LIN {X 0,Y 516.984,Z 233.939,A -85,B 0,C 180,E1 -5032.678,E2 -5032.678} C_VEL
LIN {X 0,Y 516.803,Z 243.028,A -85,B 0,C 180,E1 -5033.356,E2 -5033.356} C_VEL
LIN {X 0,Y 516.628,Z 250.94,A -85,B 0,C 180,E1 -5034.144,E2 -5034.144} C_VEL
LIN {X 0,Y 516.608,Z 257.035,A -85,B 0,C 180,E1 -5034.927,E2 -5034.927} C_VEL
LIN {X 0,Y 516.481,Z 261.852,A -85,B 0,C 180,E1 -5035.708,E2 -5035.708} C_VEL
LIN {X 0,Y 516.468,Z 265.615,A -85,B 0,C 180,E1 -5036.489,E2 -5036.489} C_VEL
LIN {X 0,Y 516.284,Z 269.666,A -85,B 0,C 180,E1 -5037.66,E2 -5037.66} C_VEL
LIN {X 0,Y 516.212,Z 271.428,A -85,B 0,C 180,E1 -5038.44,E2 -5038.44} C_VEL
LIN {X 0,Y 516.197,Z 272.491,A -85,B 0,C 180,E1 -5039.22,E2 -5039.22} C_VEL
LIN {X 0,Y 516.195,Z 272.884,A -85,B 0,C 180,E1 -5040,E2 -5040} C_VEL
LIN {X 0,Y 516.199,Z 272.616,A -85,B 0,C 180,E1 -5040.78,E2 -5040.78} C_VEL
LIN {X 0,Y 516.215,Z 271.681,A -85,B 0,C 180,E1 -5041.56,E2 -5041.56} C_VEL
LIN {X 0,Y 516.332,Z 268.959,A -85,B 0,C 180,E1 -5042.731,E2 -5042.731} C_VEL
LIN {X 0,Y 516.467,Z 266.206,A -85,B 0,C 180,E1 -5043.511,E2 -5043.511} C_VEL
LIN {X 0,Y 516.515,Z 261.551,A -85,B 0,C 180,E1 -5044.487,E2 -5044.487} C_VEL
LIN {X 0,Y 516.586,Z 256.656,A -85,B 0,C 180,E1 -5045.269,E2 -5045.269} C_VEL
LIN {X 0,Y 516.619,Z 250.449,A -85,B 0,C 180,E1 -5046.052,E2 -5046.052} C_VEL
LIN {X 0,Y 516.845,Z 242.132,A -85,B 0,C 180,E1 -5046.858,E2 -5046.858} C_VEL
LIN {X 0,Y 517.047,Z 233.07,A -85,B 0,C 180,E1 -5047.518,E2 -5047.518} C_VEL
LIN {X 0,Y 517.237,Z 222.858,A -85,B 0,C 180,E1 -5048.055,E2 -5048.055} C_VEL
LIN {X 0,Y 516.418,Z 214.88,A -85,B 0,C 180,E1 -5048.388,E2 -5048.388} C_VEL
LIN {X 0,Y 516.468,Z 207.091,A -85,B 0,C 180,E1 -5050.983,E2 -5050.983} C_VEL
LIN {X 0,Y 516.61,Z 197.576,A -85,B 0,C 180,E1 -5054.174,E2 -5054.174} C_VEL
LIN {X 0,Y 516.772,Z 188.041,A -85,B 0,C 180,E1 -5057.409,E2 -5057.409} C_VEL
LIN {X 0,Y 516.892,Z 179.78,A -85,B 0,C 180,E1 -5060.252,E2 -5060.252} C_VEL
LIN {X 0,Y 517.052,Z 171.31,A -85,B 0,C 180,E1 -5063.215,E2 -5063.215} C_VEL
LIN {X 0,Y 517.347,Z 161.729,A -85,B 0,C 180,E1 -5066.635,E2 -5066.635} C_VEL
LIN {X 0,Y 517.599,Z 153.467,A -85,B 0,C 180,E1 -5069.657,E2 -5069.657} C_VEL
LIN {X 0,Y 517.235,Z 149.681,A -85,B 0,C 180,E1 -5071.126,E2 -5071.126} C_VEL
LIN {X 0,Y 516.93,Z 148.099,A -85,B 0,C 180,E1 -5071.792,E2 -5071.792} C_VEL
LIN {X 0,Y 516.885,Z 148.104,A -85,B 0,C 180,E1 -5074.825,E2 -5074.825} C_VEL
LIN {X 0,Y 516.886,Z 148.103,A -85,B 0,C 180,E1 -5077.943,E2 -5077.943} C_VEL
LIN {X 0,Y 516.889,Z 148.101,A -85,B 0,C 180,E1 -5080.741,E2 -5080.741} C_VEL
LIN {X 0,Y 516.888,Z 148.102,A -85,B 0,C 180,E1 -5082.831,E2 -5082.831} C_VEL
LIN {X 0,Y 516.901,Z 148.1,A -85,B 0,C 180,E1 -5085.007,E2 -5085.007} C_VEL
LIN {X 0,Y 516.92,Z 148.097,A -85,B 0,C 180,E1 -5088.398,E2 -5088.398} C_VEL
LIN {X 0,Y 516.885,Z 148.103,A -85,B 0,C 180,E1 -5091.284,E2 -5091.284} C_VEL
LIN {X 0,Y 516.877,Z 148.104,A -85,B 0,C 180,E1 -5094.219,E2 -5094.219} C_VEL
LIN {X 0,Y 516.887,Z 148.104,A -85,B 0,C 180,E1 -5097.051,E2 -5097.051} C_VEL
LIN {X 0,Y 516.924,Z 148.188,A -85,B 0,C 180,E1 -5099.982,E2 -5099.982} C_VEL
LIN {X 0,Y 518.784,Z 157.254,A -85,B 0,C 180,E1 -5102.573,E2 -5102.573} C_VEL
LIN {X 0,Y 518.974,Z 160.749,A -85,B 0,C 180,E1 -5103.455,E2 -5103.455} C_VEL
LIN {X 0,Y 518.28,Z 171.627,A -85,B 0,C 180,E1 -5105.995,E2 -5105.995} C_VEL
LIN {X 0,Y 517.784,Z 182.925,A -85,B 0,C 180,E1 -5108.5,E2 -5108.5} C_VEL
LIN {X 0,Y 517.391,Z 194.575,A -85,B 0,C 180,E1 -5110.973,E2 -5110.973} C_VEL
LIN {X 0,Y 517.079,Z 207.5,A -85,B 0,C 180,E1 -5113.618,E2 -5113.618} C_VEL
LIN {X 0,Y 516.843,Z 220.945,A -85,B 0,C 180,E1 -5116.27,E2 -5116.27} C_VEL
LIN {X 0,Y 518.188,Z 232.011,A -85,B 0,C 180,E1 -5116.519,E2 -5116.519} C_VEL
LIN {X 0,Y 518.022,Z 244.633,A -85,B 0,C 180,E1 -5116.914,E2 -5116.914} C_VEL
LIN {X 0,Y 517.734,Z 256.944,A -85,B 0,C 180,E1 -5117.455,E2 -5117.455} C_VEL
LIN {X 0,Y 517.492,Z 268.95,A -85,B 0,C 180,E1 -5118.159,E2 -5118.159} C_VEL
LIN {X 0,Y 517.222,Z 280.568,A -85,B 0,C 180,E1 -5119.033,E2 -5119.033} C_VEL
LIN {X 0,Y 516.967,Z 289.07,A -85,B 0,C 180,E1 -5119.819,E2 -5119.819} C_VEL
LIN {X 0,Y 516.761,Z 297.894,A -85,B 0,C 180,E1 -5120.804,E2 -5120.804} C_VEL
LIN {X 0,Y 516.582,Z 306.427,A -85,B 0,C 180,E1 -5121.983,E2 -5121.983} C_VEL
LIN {X 0,Y 516.443,Z 312.245,A -85,B 0,C 180,E1 -5122.964,E2 -5122.964} C_VEL
LIN {X 0,Y 516.417,Z 317.908,A -85,B 0,C 180,E1 -5124.141,E2 -5124.141} C_VEL
LIN {X 0,Y 516.27,Z 322.337,A -85,B 0,C 180,E1 -5125.314,E2 -5125.314} C_VEL
LIN {X 0,Y 516.37,Z 324.685,A -85,B 0,C 180,E1 -5126.097,E2 -5126.097} C_VEL
LIN {X 0,Y 516.283,Z 326.587,A -85,B 0,C 180,E1 -5126.877,E2 -5126.877} C_VEL
LIN {X 0,Y 516.261,Z 328.016,A -85,B 0,C 180,E1 -5127.658,E2 -5127.658} C_VEL
LIN {X 0,Y 516.171,Z 329.652,A -85,B 0,C 180,E1 -5129.219,E2 -5129.219} C_VEL
LIN {X 0,Y 516.173,Z 329.879,A -85,B 0,C 180,E1 -5129.999,E2 -5129.999} C_VEL
LIN {X 0,Y 516.17,Z 329.664,A -85,B 0,C 180,E1 -5130.779,E2 -5130.779} C_VEL
LIN {X 0,Y 516.261,Z 328.056,A -85,B 0,C 180,E1 -5132.339,E2 -5132.339} C_VEL
LIN {X 0,Y 516.282,Z 326.64,A -85,B 0,C 180,E1 -5133.12,E2 -5133.12} C_VEL
LIN {X 0,Y 516.313,Z 323.669,A -85,B 0,C 180,E1 -5134.292,E2 -5134.292} C_VEL
LIN {X 0,Y 516.397,Z 319.639,A -85,B 0,C 180,E1 -5135.465,E2 -5135.465} C_VEL
LIN {X 0,Y 516.469,Z 313.671,A -85,B 0,C 180,E1 -5136.787,E2 -5136.787} C_VEL
LIN {X 0,Y 516.58,Z 306.611,A -85,B 0,C 180,E1 -5138.015,E2 -5138.015} C_VEL
LIN {X 0,Y 516.769,Z 298.141,A -85,B 0,C 180,E1 -5139.194,E2 -5139.194} C_VEL
LIN {X 0,Y 516.972,Z 289.385,A -85,B 0,C 180,E1 -5140.178,E2 -5140.178} C_VEL
LIN {X 0,Y 517.329,Z 278.602,A -85,B 0,C 180,E1 -5141.161,E2 -5141.161} C_VEL
LIN {X 0,Y 517.554,Z 267.789,A -85,B 0,C 180,E1 -5141.952,E2 -5141.952} C_VEL
LIN {X 0,Y 517.797,Z 256.672,A -85,B 0,C 180,E1 -5142.591,E2 -5142.591} C_VEL
LIN {X 0,Y 518.061,Z 244.294,A -85,B 0,C 180,E1 -5143.133,E2 -5143.133} C_VEL
LIN {X 0,Y 518.244,Z 232.51,A -85,B 0,C 180,E1 -5143.502,E2 -5143.502} C_VEL
LIN {X 0,Y 516.877,Z 220.782,A -85,B 0,C 180,E1 -5143.789,E2 -5143.789} C_VEL
LIN {X 0,Y 517.168,Z 205.909,A -85,B 0,C 180,E1 -5146.783,E2 -5146.783} C_VEL
LIN {X 0,Y 517.391,Z 194.717,A -85,B 0,C 180,E1 -5149.025,E2 -5149.025} C_VEL
LIN {X 0,Y 517.866,Z 180.952,A -85,B 0,C 180,E1 -5151.912,E2 -5151.912} C_VEL
LIN {X 0,Y 518.373,Z 167.18,A -85,B 0,C 180,E1 -5154.851,E2 -5154.851} C_VEL
LIN {X 0,Y 518.661,Z 157.378,A -85,B 0,C 180,E1 -5156.994,E2 -5156.994} C_VEL
LIN {X 0,Y 516.909,Z 148.101,A -85,B 0,C 180,E1 -5159.248,E2 -5159.248} C_VEL
LIN {X 0,Y 516.892,Z 148.102,A -85,B 0,C 180,E1 -5162.542,E2 -5162.542} C_VEL
LIN {X 0,Y 516.878,Z 148.101,A -85,B 0,C 180,E1 -5165.331,E2 -5165.331} C_VEL
LIN {X 0,Y 516.874,Z 148.101,A -85,B 0,C 180,E1 -5167.942,E2 -5167.942} C_VEL
LIN {X 0,Y 516.862,Z 148.106,A -85,B 0,C 180,E1 -5170.741,E2 -5170.741} C_VEL
LIN {X 0,Y 516.872,Z 148.102,A -85,B 0,C 180,E1 -5173.892,E2 -5173.892} C_VEL
LIN {X 0,Y 516.873,Z 148.103,A -85,B 0,C 180,E1 -5176.106,E2 -5176.106} C_VEL
LIN {X 0,Y 516.894,Z 148.101,A -85,B 0,C 180,E1 -5179.259,E2 -5179.259} C_VEL
LIN {X 0,Y 516.869,Z 148.101,A -85,B 0,C 180,E1 -5182.056,E2 -5182.056} C_VEL
LIN {X 0,Y 516.868,Z 148.099,A -85,B 0,C 180,E1 -5185.174,E2 -5185.174} C_VEL
LIN {X 0,Y 516.871,Z 148.102,A -85,B 0,C 180,E1 -5187.975,E2 -5187.975} C_VEL
LIN {X 0,Y 516.924,Z 148.097,A -85,B 0,C 180,E1 -5190.695,E2 -5190.695} C_VEL
LIN {X 0,Y 516.932,Z 148.093,A -85,B 0,C 180,E1 -5193.802,E2 -5193.802} C_VEL
LIN {X 0,Y 516.845,Z 148.102,A -85,B 0,C 180,E1 -5196.775,E2 -5196.775} C_VEL
LIN {X 0,Y 516.925,Z 148.095,A -85,B 0,C 180,E1 -5199.731,E2 -5199.731} C_VEL
LIN {X 0,Y 516.918,Z 148.098,A -85,B 0,C 180,E1 -5202.596,E2 -5202.596} C_VEL
LIN {X 0,Y 516.927,Z 148.093,A -85,B 0,C 180,E1 -5205.03,E2 -5205.03} C_VEL
LIN {X 0,Y 516.989,Z 148.085,A -85,B 0,C 180,E1 -5208.234,E2 -5208.234} C_VEL
LIN {X 0,Y 516.948,Z 148.092,A -85,B 0,C 180,E1 -5211.399,E2 -5211.399} C_VEL
LIN {X 0,Y 516.996,Z 148.084,A -85,B 0,C 180,E1 -5213.757,E2 -5213.757} C_VEL
LIN {X 0,Y 517.004,Z 148.083,A -85,B 0,C 180,E1 -5216.883,E2 -5216.883} C_VEL
LIN {X 0,Y 517.065,Z 148.076,A -85,B 0,C 180,E1 -5220,E2 -5220} C_VEL
LIN {X 0,Y 516.992,Z 148.087,A -85,B 0,C 180,E1 -5223.117,E2 -5223.117} C_VEL
LIN {X 0,Y 516.994,Z 148.089,A -85,B 0,C 180,E1 -5226.243,E2 -5226.243} C_VEL
LIN {X 0,Y 516.946,Z 148.095,A -85,B 0,C 180,E1 -5229.389,E2 -5229.389} C_VEL
LIN {X 0,Y 516.968,Z 148.088,A -85,B 0,C 180,E1 -5231.824,E2 -5231.824} C_VEL
LIN {X 0,Y 516.931,Z 148.092,A -85,B 0,C 180,E1 -5235.148,E2 -5235.148} C_VEL
LIN {X 0,Y 516.911,Z 148.098,A -85,B 0,C 180,E1 -5238.223,E2 -5238.223} C_VEL
LIN {X 0,Y 516.901,Z 148.097,A -85,B 0,C 180,E1 -5240.702,E2 -5240.702} C_VEL
LIN {X 0,Y 516.878,Z 148.102,A -85,B 0,C 180,E1 -5243.223,E2 -5243.223} C_VEL
LIN {X 0,Y 516.888,Z 148.102,A -85,B 0,C 180,E1 -5246.188,E2 -5246.188} C_VEL
LIN {X 0,Y 516.903,Z 148.099,A -85,B 0,C 180,E1 -5249.526,E2 -5249.526} C_VEL
LIN {X 0,Y 516.889,Z 148.099,A -85,B 0,C 180,E1 -5252.545,E2 -5252.545} C_VEL
LIN {X 0,Y 516.872,Z 148.1,A -85,B 0,C 180,E1 -5255.334,E2 -5255.334} C_VEL
LIN {X 0,Y 516.868,Z 148.105,A -85,B 0,C 180,E1 -5257.944,E2 -5257.944} C_VEL
LIN {X 0,Y 516.871,Z 148.098,A -85,B 0,C 180,E1 -5260.743,E2 -5260.743} C_VEL
LIN {X 0,Y 516.874,Z 148.102,A -85,B 0,C 180,E1 -5262.832,E2 -5262.832} C_VEL
LIN {X 0,Y 516.913,Z 148.099,A -85,B 0,C 180,E1 -5265.011,E2 -5265.011} C_VEL
LIN {X 0,Y 516.909,Z 148.099,A -85,B 0,C 180,E1 -5268.4,E2 -5268.4} C_VEL
LIN {X 0,Y 516.872,Z 148.1,A -85,B 0,C 180,E1 -5270.322,E2 -5270.322} C_VEL
LIN {X 0,Y 516.198,Z 148.185,A -85,B 0,C 180,E1 -5270.972,E2 -5270.972} C_VEL
LIN {X 0,Y 513.338,Z 148.54,A -85,B 0,C 180,E1 -5272.027,E2 -5272.027} C_VEL
LIN {X 0,Y 510.923,Z 148.842,A -85,B 0,C 180,E1 -5272.878,E2 -5272.878} C_VEL
LIN {X 0,Y 509.883,Z 148.972,A -85,B 0,C 180,E1 -5273.534,E2 -5273.534} C_VEL
LIN {X 0,Y 509.797,Z 148.981,A -85,B 0,C 180,E1 -5273.757,E2 -5273.757} C_VEL
LIN {X 0,Y 509.853,Z 148.978,A -85,B 0,C 180,E1 -5276.541,E2 -5276.541} C_VEL
LIN {X 0,Y 509.845,Z 148.976,A -85,B 0,C 180,E1 -5279.336,E2 -5279.336} C_VEL
LIN {X 0,Y 509.89,Z 148.971,A -85,B 0,C 180,E1 -5282.056,E2 -5282.056} C_VEL
LIN {X 0,Y 509.806,Z 148.983,A -85,B 0,C 180,E1 -5284.702,E2 -5284.702} C_VEL
LIN {X 0,Y 509.82,Z 148.977,A -85,B 0,C 180,E1 -5287.46,E2 -5287.46} C_VEL
LIN {X 0,Y 509.914,Z 148.97,A -85,B 0,C 180,E1 -5289.846,E2 -5289.846} C_VEL
LIN {X 0,Y 509.883,Z 148.975,A -85,B 0,C 180,E1 -5293.176,E2 -5293.176} C_VEL
LIN {X 0,Y 509.852,Z 148.974,A -85,B 0,C 180,E1 -5295.635,E2 -5295.635} C_VEL
LIN {X 0,Y 509.911,Z 148.967,A -85,B 0,C 180,E1 -5298.876,E2 -5298.876} C_VEL
LIN {X 0,Y 509.951,Z 148.964,A -85,B 0,C 180,E1 -5302.08,E2 -5302.08} C_VEL
LIN {X 0,Y 509.983,Z 148.959,A -85,B 0,C 180,E1 -5304.466,E2 -5304.466} C_VEL
LIN {X 0,Y 510.056,Z 148.949,A -85,B 0,C 180,E1 -5307.632,E2 -5307.632} C_VEL
LIN {X 0,Y 510.036,Z 148.956,A -85,B 0,C 180,E1 -5310.001,E2 -5310.001} C_VEL
LIN {X 0,Y 510.051,Z 148.949,A -85,B 0,C 180,E1 -5312.37,E2 -5312.37} C_VEL
LIN {X 0,Y 509.982,Z 148.959,A -85,B 0,C 180,E1 -5316.331,E2 -5316.331} C_VEL
LIN {X 0,Y 509.914,Z 148.97,A -85,B 0,C 180,E1 -5318.721,E2 -5318.721} C_VEL
LIN {X 0,Y 509.908,Z 148.971,A -85,B 0,C 180,E1 -5321.933,E2 -5321.933} C_VEL
LIN {X 0,Y 509.899,Z 148.973,A -85,B 0,C 180,E1 -5325.243,E2 -5325.243} C_VEL
LIN {X 0,Y 509.866,Z 148.976,A -85,B 0,C 180,E1 -5328.485,E2 -5328.485} C_VEL
LIN {X 0,Y 509.855,Z 148.974,A -85,B 0,C 180,E1 -5331.003,E2 -5331.003} C_VEL
LIN {X 0,Y 509.822,Z 148.983,A -85,B 0,C 180,E1 -5333.565,E2 -5333.565} C_VEL
LIN {X 0,Y 509.819,Z 148.977,A -85,B 0,C 180,E1 -5336.357,E2 -5336.357} C_VEL
LIN {X 0,Y 509.842,Z 148.979,A -85,B 0,C 180,E1 -5338.847,E2 -5338.847} C_VEL
LIN {X 0,Y 509.823,Z 148.98,A -85,B 0,C 180,E1 -5341.591,E2 -5341.591} C_VEL
LIN {X 0,Y 509.843,Z 148.976,A -85,B 0,C 180,E1 -5344.415,E2 -5344.415} C_VEL
LIN {X 0,Y 509.793,Z 148.983,A -85,B 0,C 180,E1 -5347.344,E2 -5347.344} C_VEL
LIN {X 0,Y 509.818,Z 148.983,A -85,B 0,C 180,E1 -5350.385,E2 -5350.385} C_VEL
LIN {X 0,Y 509.808,Z 148.98,A -85,B 0,C 180,E1 -5353.06,E2 -5353.06} C_VEL
LIN {X 0,Y 509.828,Z 148.98,A -85,B 0,C 180,E1 -5355.794,E2 -5355.794} C_VEL
LIN {X 0,Y 509.86,Z 148.977,A -85,B 0,C 180,E1 -5358.575,E2 -5358.575} C_VEL
LIN {X 0,Y 509.819,Z 148.979,A -85,B 0,C 180,E1 -5361.792,E2 -5361.792} C_VEL
LIN {X 0,Y 509.83,Z 148.977,A -85,B 0,C 180,E1 -5364.622,E2 -5364.622} C_VEL
LIN {X 0,Y 509.865,Z 148.977,A -85,B 0,C 180,E1 -5367.481,E2 -5367.481} C_VEL
LIN {X 0,Y 509.905,Z 149.045,A -85,B 0,C 180,E1 -5368.71,E2 -5368.71} C_VEL
LIN {X 0,Y 510.39,Z 153.219,A -85,B 0,C 180,E1 -5370.283,E2 -5370.283} C_VEL
LIN {X 0,Y 510.177,Z 162.264,A -85,B 0,C 180,E1 -5373.563,E2 -5373.563} C_VEL
LIN {X 0,Y 509.935,Z 170.358,A -85,B 0,C 180,E1 -5376.442,E2 -5376.442} C_VEL
LIN {X 0,Y 509.805,Z 179.405,A -85,B 0,C 180,E1 -5379.625,E2 -5379.625} C_VEL
LIN {X 0,Y 509.665,Z 188.47,A -85,B 0,C 180,E1 -5382.754,E2 -5382.754} C_VEL
LIN {X 0,Y 509.53,Z 196.847,A -85,B 0,C 180,E1 -5385.625,E2 -5385.625} C_VEL
LIN {X 0,Y 509.379,Z 206.394,A -85,B 0,C 180,E1 -5388.863,E2 -5388.863} C_VEL
LIN {X 0,Y 509.323,Z 214.658,A -85,B 0,C 180,E1 -5391.619,E2 -5391.619} C_VEL
LIN {X 0,Y 510.161,Z 224.625,A -85,B 0,C 180,E1 -5392.032,E2 -5392.032} C_VEL
LIN {X 0,Y 509.982,Z 234.394,A -85,B 0,C 180,E1 -5392.577,E2 -5392.577} C_VEL
LIN {X 0,Y 509.761,Z 243.417,A -85,B 0,C 180,E1 -5393.264,E2 -5393.264} C_VEL
LIN {X 0,Y 509.571,Z 251.31,A -85,B 0,C 180,E1 -5394.063,E2 -5394.063} C_VEL
LIN {X 0,Y 509.555,Z 257.394,A -85,B 0,C 180,E1 -5394.857,E2 -5394.857} C_VEL
LIN {X 0,Y 509.423,Z 262.208,A -85,B 0,C 180,E1 -5395.648,E2 -5395.648} C_VEL
LIN {X 0,Y 509.41,Z 265.977,A -85,B 0,C 180,E1 -5396.441,E2 -5396.441} C_VEL
LIN {X 0,Y 509.215,Z 270.043,A -85,B 0,C 180,E1 -5397.627,E2 -5397.627} C_VEL
LIN {X 0,Y 509.132,Z 271.812,A -85,B 0,C 180,E1 -5398.418,E2 -5398.418} C_VEL
LIN {X 0,Y 509.109,Z 272.882,A -85,B 0,C 180,E1 -5399.209,E2 -5399.209} C_VEL
LIN {X 0,Y 509.107,Z 273.28,A -85,B 0,C 180,E1 -5400,E2 -5400} C_VEL
LIN {X 0,Y 509.111,Z 273.015,A -85,B 0,C 180,E1 -5400.791,E2 -5400.791} C_VEL
LIN {X 0,Y 509.135,Z 272.081,A -85,B 0,C 180,E1 -5401.582,E2 -5401.582} C_VEL
LIN {X 0,Y 509.265,Z 269.368,A -85,B 0,C 180,E1 -5402.769,E2 -5402.769} C_VEL
LIN {X 0,Y 509.433,Z 264.916,A -85,B 0,C 180,E1 -5403.955,E2 -5403.955} C_VEL
LIN {X 0,Y 509.539,Z 259.653,A -85,B 0,C 180,E1 -5404.945,E2 -5404.945} C_VEL
LIN {X 0,Y 509.612,Z 254.178,A -85,B 0,C 180,E1 -5405.738,E2 -5405.738} C_VEL
LIN {X 0,Y 509.717,Z 247.409,A -85,B 0,C 180,E1 -5406.508,E2 -5406.508} C_VEL
LIN {X 0,Y 509.902,Z 239.278,A -85,B 0,C 180,E1 -5407.225,E2 -5407.225} C_VEL
LIN {X 0,Y 510.131,Z 230.408,A -85,B 0,C 180,E1 -5407.819,E2 -5407.819} C_VEL
LIN {X 0,Y 510.108,Z 221.392,A -85,B 0,C 180,E1 -5408.268,E2 -5408.268} C_VEL
LIN {X 0,Y 509.353,Z 215.03,A -85,B 0,C 180,E1 -5408.53,E2 -5408.53} C_VEL
LIN {X 0,Y 509.411,Z 207.298,A -85,B 0,C 180,E1 -5411.137,E2 -5411.137} C_VEL
LIN {X 0,Y 509.55,Z 198.944,A -85,B 0,C 180,E1 -5413.968,E2 -5413.968} C_VEL
LIN {X 0,Y 509.684,Z 190.62,A -85,B 0,C 180,E1 -5416.832,E2 -5416.832} C_VEL
LIN {X 0,Y 509.854,Z 182.264,A -85,B 0,C 180,E1 -5419.738,E2 -5419.738} C_VEL
LIN {X 0,Y 510.02,Z 173.92,A -85,B 0,C 180,E1 -5422.696,E2 -5422.696} C_VEL
LIN {X 0,Y 510.222,Z 165.574,A -85,B 0,C 180,E1 -5425.715,E2 -5425.715} C_VEL
LIN {X 0,Y 510.576,Z 157.23,A -85,B 0,C 180,E1 -5428.801,E2 -5428.801} C_VEL
LIN {X 0,Y 510.506,Z 152.507,A -85,B 0,C 180,E1 -5430.622,E2 -5430.622} C_VEL
LIN {X 0,Y 509.857,Z 148.98,A -85,B 0,C 180,E1 -5432.169,E2 -5432.169} C_VEL
LIN {X 0,Y 509.835,Z 148.981,A -85,B 0,C 180,E1 -5435.378,E2 -5435.378} C_VEL
LIN {X 0,Y 509.855,Z 148.978,A -85,B 0,C 180,E1 -5438.338,E2 -5438.338} C_VEL
LIN {X 0,Y 509.861,Z 148.978,A -85,B 0,C 180,E1 -5441.425,E2 -5441.425} C_VEL
LIN {X 0,Y 509.845,Z 148.98,A -85,B 0,C 180,E1 -5444.67,E2 -5444.67} C_VEL
LIN {X 0,Y 509.839,Z 148.979,A -85,B 0,C 180,E1 -5447.51,E2 -5447.51} C_VEL
LIN {X 0,Y 509.851,Z 148.978,A -85,B 0,C 180,E1 -5450.647,E2 -5450.647} C_VEL
LIN {X 0,Y 509.831,Z 148.982,A -85,B 0,C 180,E1 -5453.646,E2 -5453.646} C_VEL
LIN {X 0,Y 509.848,Z 148.98,A -85,B 0,C 180,E1 -5456.537,E2 -5456.537} C_VEL
LIN {X 0,Y 509.873,Z 149.1,A -85,B 0,C 180,E1 -5459.565,E2 -5459.565} C_VEL
LIN {X 0,Y 511.72,Z 157.754,A -85,B 0,C 180,E1 -5462.162,E2 -5462.162} C_VEL
LIN {X 0,Y 512.12,Z 161.356,A -85,B 0,C 180,E1 -5463.128,E2 -5463.128} C_VEL
LIN {X 0,Y 511.433,Z 171.788,A -85,B 0,C 180,E1 -5465.653,E2 -5465.653} C_VEL
LIN {X 0,Y 510.78,Z 184.859,A -85,B 0,C 180,E1 -5468.615,E2 -5468.615} C_VEL
LIN {X 0,Y 510.299,Z 199.961,A -85,B 0,C 180,E1 -5471.859,E2 -5471.859} C_VEL
LIN {X 0,Y 509.878,Z 215.321,A -85,B 0,C 180,E1 -5475.021,E2 -5475.021} C_VEL
LIN {X 0,Y 509.822,Z 220.716,A -85,B 0,C 180,E1 -5476.115,E2 -5476.115} C_VEL
LIN {X 0,Y 511.155,Z 233.061,A -85,B 0,C 180,E1 -5476.406,E2 -5476.406} C_VEL
LIN {X 0,Y 510.997,Z 245.969,A -85,B 0,C 180,E1 -5476.832,E2 -5476.832} C_VEL
LIN {X 0,Y 510.713,Z 257.682,A -85,B 0,C 180,E1 -5477.369,E2 -5477.369} C_VEL
LIN {X 0,Y 510.441,Z 269.393,A -85,B 0,C 180,E1 -5478.08,E2 -5478.08} C_VEL
LIN {X 0,Y 510.161,Z 279.855,A -85,B 0,C 180,E1 -5478.879,E2 -5478.879} C_VEL
LIN {X 0,Y 509.864,Z 290.385,A -85,B 0,C 180,E1 -5479.877,E2 -5479.877} C_VEL
LIN {X 0,Y 509.652,Z 298.879,A -85,B 0,C 180,E1 -5480.874,E2 -5480.874} C_VEL
LIN {X 0,Y 509.49,Z 307.166,A -85,B 0,C 180,E1 -5482.07,E2 -5482.07} C_VEL
LIN {X 0,Y 509.308,Z 314.019,A -85,B 0,C 180,E1 -5483.303,E2 -5483.303} C_VEL
LIN {X 0,Y 509.309,Z 319.096,A -85,B 0,C 180,E1 -5484.456,E2 -5484.456} C_VEL
LIN {X 0,Y 509.221,Z 323.171,A -85,B 0,C 180,E1 -5485.645,E2 -5485.645} C_VEL
LIN {X 0,Y 509.202,Z 326.178,A -85,B 0,C 180,E1 -5486.834,E2 -5486.834} C_VEL
LIN {X 0,Y 509.19,Z 327.617,A -85,B 0,C 180,E1 -5487.626,E2 -5487.626} C_VEL
LIN {X 0,Y 509.084,Z 329.262,A -85,B 0,C 180,E1 -5489.208,E2 -5489.208} C_VEL
LIN {X 0,Y 509.084,Z 329.492,A -85,B 0,C 180,E1 -5489.999,E2 -5489.999} C_VEL
LIN {X 0,Y 509.112,Z 328.668,A -85,B 0,C 180,E1 -5491.581,E2 -5491.581} C_VEL
LIN {X 0,Y 509.19,Z 327.67,A -85,B 0,C 180,E1 -5492.372,E2 -5492.372} C_VEL
LIN {X 0,Y 509.201,Z 326.247,A -85,B 0,C 180,E1 -5493.164,E2 -5493.164} C_VEL
LIN {X 0,Y 509.206,Z 323.267,A -85,B 0,C 180,E1 -5494.352,E2 -5494.352} C_VEL
LIN {X 0,Y 509.309,Z 319.223,A -85,B 0,C 180,E1 -5495.542,E2 -5495.542} C_VEL
LIN {X 0,Y 509.399,Z 313.075,A -85,B 0,C 180,E1 -5496.912,E2 -5496.912} C_VEL
LIN {X 0,Y 509.496,Z 306.149,A -85,B 0,C 180,E1 -5498.127,E2 -5498.127} C_VEL
LIN {X 0,Y 509.717,Z 297.628,A -85,B 0,C 180,E1 -5499.322,E2 -5499.322} C_VEL
LIN {X 0,Y 509.945,Z 288.829,A -85,B 0,C 180,E1 -5500.32,E2 -5500.32} C_VEL
LIN {X 0,Y 510.317,Z 277.992,A -85,B 0,C 180,E1 -5501.316,E2 -5501.316} C_VEL
LIN {X 0,Y 510.505,Z 267.095,A -85,B 0,C 180,E1 -5502.116,E2 -5502.116} C_VEL
LIN {X 0,Y 510.817,Z 254.81,A -85,B 0,C 180,E1 -5502.816,E2 -5502.816} C_VEL
LIN {X 0,Y 511.111,Z 241.903,A -85,B 0,C 180,E1 -5503.365,E2 -5503.365} C_VEL
LIN {X 0,Y 511.158,Z 231.034,A -85,B 0,C 180,E1 -5503.693,E2 -5503.693} C_VEL
LIN {X 0,Y 509.846,Z 220.799,A -85,B 0,C 180,E1 -5503.932,E2 -5503.932} C_VEL
LIN {X 0,Y 510.194,Z 204.761,A -85,B 0,C 180,E1 -5507.226,E2 -5507.226} C_VEL
LIN {X 0,Y 510.485,Z 192.708,A -85,B 0,C 180,E1 -5509.711,E2 -5509.711} C_VEL
LIN {X 0,Y 511.056,Z 177.902,A -85,B 0,C 180,E1 -5512.871,E2 -5512.871} C_VEL
LIN {X 0,Y 511.586,Z 165.203,A -85,B 0,C 180,E1 -5515.64,E2 -5515.64} C_VEL
LIN {X 0,Y 511.769,Z 159.354,A -85,B 0,C 180,E1 -5516.946,E2 -5516.946} C_VEL
LIN {X 0,Y 510.367,Z 151.552,A -85,B 0,C 180,E1 -5518.812,E2 -5518.812} C_VEL
LIN {X 0,Y 509.871,Z 148.977,A -85,B 0,C 180,E1 -5519.455,E2 -5519.455} C_VEL
LIN {X 0,Y 509.869,Z 148.975,A -85,B 0,C 180,E1 -5522.773,E2 -5522.773} C_VEL
LIN {X 0,Y 509.837,Z 148.981,A -85,B 0,C 180,E1 -5525.58,E2 -5525.58} C_VEL
LIN {X 0,Y 509.842,Z 148.975,A -85,B 0,C 180,E1 -5528.337,E2 -5528.337} C_VEL
LIN {X 0,Y 509.836,Z 148.975,A -85,B 0,C 180,E1 -5531.425,E2 -5531.425} C_VEL
LIN {X 0,Y 509.847,Z 148.976,A -85,B 0,C 180,E1 -5534.667,E2 -5534.667} C_VEL
LIN {X 0,Y 509.854,Z 148.975,A -85,B 0,C 180,E1 -5538.101,E2 -5538.101} C_VEL
LIN {X 0,Y 509.866,Z 148.976,A -85,B 0,C 180,E1 -5540.649,E2 -5540.649} C_VEL
LIN {X 0,Y 509.796,Z 148.981,A -85,B 0,C 180,E1 -5543.644,E2 -5543.644} C_VEL
LIN {X 0,Y 509.847,Z 148.975,A -85,B 0,C 180,E1 -5546.538,E2 -5546.538} C_VEL
LIN {X 0,Y 509.839,Z 148.98,A -85,B 0,C 180,E1 -5549.334,E2 -5549.334} C_VEL
LIN {X 0,Y 509.883,Z 148.971,A -85,B 0,C 180,E1 -5552.054,E2 -5552.054} C_VEL
LIN {X 0,Y 509.86,Z 148.974,A -85,B 0,C 180,E1 -5554.703,E2 -5554.703} C_VEL
LIN {X 0,Y 509.811,Z 148.982,A -85,B 0,C 180,E1 -5557.457,E2 -5557.457} C_VEL
LIN {X 0,Y 509.903,Z 148.969,A -85,B 0,C 180,E1 -5559.844,E2 -5559.844} C_VEL
LIN {X 0,Y 509.874,Z 148.973,A -85,B 0,C 180,E1 -5563.174,E2 -5563.174} C_VEL
LIN {X 0,Y 509.851,Z 148.976,A -85,B 0,C 180,E1 -5565.634,E2 -5565.634} C_VEL
LIN {X 0,Y 509.903,Z 148.968,A -85,B 0,C 180,E1 -5568.874,E2 -5568.874} C_VEL
LIN {X 0,Y 509.934,Z 148.964,A -85,B 0,C 180,E1 -5572.078,E2 -5572.078} C_VEL
LIN {X 0,Y 509.979,Z 148.962,A -85,B 0,C 180,E1 -5574.464,E2 -5574.464} C_VEL
LIN {X 0,Y 510.042,Z 148.955,A -85,B 0,C 180,E1 -5577.631,E2 -5577.631} C_VEL
LIN {X 0,Y 510.036,Z 148.952,A -85,B 0,C 180,E1 -5580,E2 -5580} C_VEL
LIN {X 0,Y 510.031,Z 148.952,A -85,B 0,C 180,E1 -5582.369,E2 -5582.369} C_VEL
LIN {X 0,Y 509.963,Z 148.965,A -85,B 0,C 180,E1 -5586.33,E2 -5586.33} C_VEL
LIN {X 0,Y 509.906,Z 148.968,A -85,B 0,C 180,E1 -5588.72,E2 -5588.72} C_VEL
LIN {X 0,Y 509.936,Z 148.964,A -85,B 0,C 180,E1 -5591.931,E2 -5591.931} C_VEL
LIN {X 0,Y 509.878,Z 148.97,A -85,B 0,C 180,E1 -5595.242,E2 -5595.242} C_VEL
LIN {X 0,Y 509.874,Z 148.976,A -85,B 0,C 180,E1 -5598.002,E2 -5598.002} C_VEL
LIN {X 0,Y 509.844,Z 148.978,A -85,B 0,C 180,E1 -5601.002,E2 -5601.002} C_VEL
LIN {X 0,Y 509.837,Z 148.977,A -85,B 0,C 180,E1 -5603.563,E2 -5603.563} C_VEL
LIN {X 0,Y 509.864,Z 148.977,A -85,B 0,C 180,E1 -5606.372,E2 -5606.372} C_VEL
LIN {X 0,Y 509.845,Z 148.98,A -85,B 0,C 180,E1 -5609.752,E2 -5609.752} C_VEL
LIN {X 0,Y 509.865,Z 148.976,A -85,B 0,C 180,E1 -5612.776,E2 -5612.776} C_VEL
LIN {X 0,Y 509.832,Z 148.977,A -85,B 0,C 180,E1 -5615.582,E2 -5615.582} C_VEL
LIN {X 0,Y 509.838,Z 148.978,A -85,B 0,C 180,E1 -5618.339,E2 -5618.339} C_VEL
LIN {X 0,Y 509.844,Z 148.98,A -85,B 0,C 180,E1 -5621.427,E2 -5621.427} C_VEL
LIN {X 0,Y 509.847,Z 148.978,A -85,B 0,C 180,E1 -5624.669,E2 -5624.669} C_VEL
LIN {X 0,Y 509.852,Z 148.978,A -85,B 0,C 180,E1 -5628.104,E2 -5628.104} C_VEL
LIN {X 0,Y 509.837,Z 148.976,A -85,B 0,C 180,E1 -5630.649,E2 -5630.649} C_VEL
LIN {X 0,Y 509.797,Z 148.981,A -85,B 0,C 180,E1 -5633.757,E2 -5633.757} C_VEL
LIN {X 0,Y 509.139,Z 149.064,A -85,B 0,C 180,E1 -5634.417,E2 -5634.417} C_VEL
LIN {X 0,Y 506.331,Z 149.413,A -85,B 0,C 180,E1 -5635.489,E2 -5635.489} C_VEL
LIN {X 0,Y 503.943,Z 149.713,A -85,B 0,C 180,E1 -5636.353,E2 -5636.353} C_VEL
LIN {X 0,Y 502.898,Z 149.842,A -85,B 0,C 180,E1 -5637.019,E2 -5637.019} C_VEL
LIN {X 0,Y 502.802,Z 149.853,A -85,B 0,C 180,E1 -5637.245,E2 -5637.245} C_VEL
LIN {X 0,Y 502.825,Z 149.853,A -85,B 0,C 180,E1 -5640.063,E2 -5640.063} C_VEL
LIN {X 0,Y 502.826,Z 149.849,A -85,B 0,C 180,E1 -5642.535,E2 -5642.535} C_VEL
LIN {X 0,Y 502.767,Z 149.857,A -85,B 0,C 180,E1 -5645.314,E2 -5645.314} C_VEL
LIN {X 0,Y 502.776,Z 149.856,A -85,B 0,C 180,E1 -5647.828,E2 -5647.828} C_VEL
LIN {X 0,Y 502.823,Z 149.852,A -85,B 0,C 180,E1 -5650.402,E2 -5650.402} C_VEL
LIN {X 0,Y 502.832,Z 149.851,A -85,B 0,C 180,E1 -5652.933,E2 -5652.933} C_VEL
LIN {X 0,Y 502.836,Z 149.849,A -85,B 0,C 180,E1 -5655.43,E2 -5655.43} C_VEL
LIN {X 0,Y 502.875,Z 149.844,A -85,B 0,C 180,E1 -5658.718,E2 -5658.718} C_VEL
LIN {X 0,Y 502.901,Z 149.844,A -85,B 0,C 180,E1 -5661.968,E2 -5661.968} C_VEL
LIN {X 0,Y 502.939,Z 149.836,A -85,B 0,C 180,E1 -5664.388,E2 -5664.388} C_VEL
LIN {X 0,Y 503.026,Z 149.824,A -85,B 0,C 180,E1 -5667.599,E2 -5667.599} C_VEL
LIN {X 0,Y 503.005,Z 149.831,A -85,B 0,C 180,E1 -5670.001,E2 -5670.001} C_VEL
LIN {X 0,Y 503.02,Z 149.825,A -85,B 0,C 180,E1 -5672.403,E2 -5672.403} C_VEL
LIN {X 0,Y 502.939,Z 149.837,A -85,B 0,C 180,E1 -5675.615,E2 -5675.615} C_VEL
LIN {X 0,Y 502.904,Z 149.841,A -85,B 0,C 180,E1 -5678.034,E2 -5678.034} C_VEL
LIN {X 0,Y 502.88,Z 149.843,A -85,B 0,C 180,E1 -5681.284,E2 -5681.284} C_VEL
LIN {X 0,Y 502.827,Z 149.848,A -85,B 0,C 180,E1 -5684.572,E2 -5684.572} C_VEL
LIN {X 0,Y 502.822,Z 149.854,A -85,B 0,C 180,E1 -5687.07,E2 -5687.07} C_VEL
LIN {X 0,Y 502.828,Z 149.85,A -85,B 0,C 180,E1 -5689.601,E2 -5689.601} C_VEL
LIN {X 0,Y 502.806,Z 149.852,A -85,B 0,C 180,E1 -5692.703,E2 -5692.703} C_VEL
LIN {X 0,Y 502.78,Z 149.855,A -85,B 0,C 180,E1 -5695.68,E2 -5695.68} C_VEL
LIN {X 0,Y 502.778,Z 149.857,A -85,B 0,C 180,E1 -5698.378,E2 -5698.378} C_VEL
LIN {X 0,Y 502.797,Z 149.853,A -85,B 0,C 180,E1 -5701.144,E2 -5701.144} C_VEL
LIN {X 0,Y 502.794,Z 149.856,A -85,B 0,C 180,E1 -5703.996,E2 -5703.996} C_VEL
LIN {X 0,Y 502.754,Z 149.861,A -85,B 0,C 180,E1 -5707.174,E2 -5707.174} C_VEL
LIN {X 0,Y 502.773,Z 149.857,A -85,B 0,C 180,E1 -5710.018,E2 -5710.018} C_VEL
LIN {X 0,Y 502.779,Z 149.86,A -85,B 0,C 180,E1 -5712.196,E2 -5712.196} C_VEL
LIN {X 0,Y 502.791,Z 149.857,A -85,B 0,C 180,E1 -5715.471,E2 -5715.471} C_VEL
LIN {X 0,Y 502.825,Z 149.852,A -85,B 0,C 180,E1 -5718.934,E2 -5718.934} C_VEL
LIN {X 0,Y 502.768,Z 149.86,A -85,B 0,C 180,E1 -5722.044,E2 -5722.044} C_VEL
LIN {X 0,Y 502.798,Z 149.854,A -85,B 0,C 180,E1 -5725.034,E2 -5725.034} C_VEL
LIN {X 0,Y 502.81,Z 149.854,A -85,B 0,C 180,E1 -5727.917,E2 -5727.917} C_VEL
LIN {X 0,Y 502.884,Z 149.998,A -85,B 0,C 180,E1 -5728.623,E2 -5728.623} C_VEL
LIN {X 0,Y 503.366,Z 154.553,A -85,B 0,C 180,E1 -5730.355,E2 -5730.355} C_VEL
LIN {X 0,Y 503.161,Z 163.009,A -85,B 0,C 180,E1 -5733.451,E2 -5733.451} C_VEL
LIN {X 0,Y 502.953,Z 170.334,A -85,B 0,C 180,E1 -5736.094,E2 -5736.094} C_VEL
LIN {X 0,Y 502.759,Z 180.052,A -85,B 0,C 180,E1 -5739.545,E2 -5739.545} C_VEL
LIN {X 0,Y 502.599,Z 188.491,A -85,B 0,C 180,E1 -5742.504,E2 -5742.504} C_VEL
LIN {X 0,Y 502.474,Z 196.938,A -85,B 0,C 180,E1 -5745.418,E2 -5745.418} C_VEL
LIN {X 0,Y 502.331,Z 206.538,A -85,B 0,C 180,E1 -5748.704,E2 -5748.704} C_VEL
LIN {X 0,Y 502.228,Z 214.728,A -85,B 0,C 180,E1 -5751.475,E2 -5751.475} C_VEL
LIN {X 0,Y 503.179,Z 224.133,A -85,B 0,C 180,E1 -5751.87,E2 -5751.87} C_VEL
LIN {X 0,Y 502.973,Z 233.305,A -85,B 0,C 180,E1 -5752.372,E2 -5752.372} C_VEL
LIN {X 0,Y 502.789,Z 241.303,A -85,B 0,C 180,E1 -5752.954,E2 -5752.954} C_VEL
LIN {X 0,Y 502.567,Z 249.904,A -85,B 0,C 180,E1 -5753.778,E2 -5753.778} C_VEL
LIN {X 0,Y 502.493,Z 256.37,A -85,B 0,C 180,E1 -5754.583,E2 -5754.583} C_VEL
LIN {X 0,Y 502.37,Z 262.564,A -85,B 0,C 180,E1 -5755.587,E2 -5755.587} C_VEL
LIN {X 0,Y 502.353,Z 266.338,A -85,B 0,C 180,E1 -5756.391,E2 -5756.391} C_VEL
LIN {X 0,Y 502.149,Z 270.42,A -85,B 0,C 180,E1 -5757.594,E2 -5757.594} C_VEL
LIN {X 0,Y 502.055,Z 272.196,A -85,B 0,C 180,E1 -5758.396,E2 -5758.396} C_VEL
LIN {X 0,Y 502.024,Z 273.272,A -85,B 0,C 180,E1 -5759.198,E2 -5759.198} C_VEL
LIN {X 0,Y 502.02,Z 273.676,A -85,B 0,C 180,E1 -5760,E2 -5760} C_VEL
LIN {X 0,Y 502.026,Z 273.414,A -85,B 0,C 180,E1 -5760.802,E2 -5760.802} C_VEL
LIN {X 0,Y 502.058,Z 272.482,A -85,B 0,C 180,E1 -5761.604,E2 -5761.604} C_VEL
LIN {X 0,Y 502.201,Z 269.773,A -85,B 0,C 180,E1 -5762.808,E2 -5762.808} C_VEL
LIN {X 0,Y 502.356,Z 267.014,A -85,B 0,C 180,E1 -5763.61,E2 -5763.61} C_VEL
LIN {X 0,Y 502.423,Z 262.376,A -85,B 0,C 180,E1 -5764.613,E2 -5764.613} C_VEL
LIN {X 0,Y 502.462,Z 256.104,A -85,B 0,C 180,E1 -5765.619,E2 -5765.619} C_VEL
LIN {X 0,Y 502.635,Z 249.572,A -85,B 0,C 180,E1 -5766.423,E2 -5766.423} C_VEL
LIN {X 0,Y 502.854,Z 241.086,A -85,B 0,C 180,E1 -5767.226,E2 -5767.226} C_VEL
LIN {X 0,Y 503.132,Z 232.756,A -85,B 0,C 180,E1 -5767.828,E2 -5767.828} C_VEL
LIN {X 0,Y 503.242,Z 223.478,A -85,B 0,C 180,E1 -5768.331,E2 -5768.331} C_VEL
LIN {X 0,Y 502.284,Z 215.105,A -85,B 0,C 180,E1 -5768.702,E2 -5768.702} C_VEL
LIN {X 0,Y 502.394,Z 206.328,A -85,B 0,C 180,E1 -5771.695,E2 -5771.695} C_VEL
LIN {X 0,Y 502.551,Z 197.972,A -85,B 0,C 180,E1 -5774.58,E2 -5774.58} C_VEL
LIN {X 0,Y 502.715,Z 188.443,A -85,B 0,C 180,E1 -5777.912,E2 -5777.912} C_VEL
LIN {X 0,Y 502.897,Z 180.106,A -85,B 0,C 180,E1 -5780.877,E2 -5780.877} C_VEL
LIN {X 0,Y 503.067,Z 171.79,A -85,B 0,C 180,E1 -5783.9,E2 -5783.9} C_VEL
LIN {X 0,Y 503.404,Z 163.418,A -85,B 0,C 180,E1 -5787.002,E2 -5787.002} C_VEL
LIN {X 0,Y 503.716,Z 156.473,A -85,B 0,C 180,E1 -5789.664,E2 -5789.664} C_VEL
LIN {X 0,Y 503.223,Z 151.805,A -85,B 0,C 180,E1 -5791.577,E2 -5791.577} C_VEL
LIN {X 0,Y 502.834,Z 149.855,A -85,B 0,C 180,E1 -5792.436,E2 -5792.436} C_VEL
LIN {X 0,Y 502.801,Z 149.858,A -85,B 0,C 180,E1 -5794.966,E2 -5794.966} C_VEL
LIN {X 0,Y 502.799,Z 149.857,A -85,B 0,C 180,E1 -5797.954,E2 -5797.954} C_VEL
LIN {X 0,Y 502.825,Z 149.853,A -85,B 0,C 180,E1 -5801.066,E2 -5801.066} C_VEL
LIN {X 0,Y 502.792,Z 149.858,A -85,B 0,C 180,E1 -5804.53,E2 -5804.53} C_VEL
LIN {X 0,Y 502.802,Z 149.857,A -85,B 0,C 180,E1 -5807.86,E2 -5807.86} C_VEL
LIN {X 0,Y 502.807,Z 149.857,A -85,B 0,C 180,E1 -5811.023,E2 -5811.023} C_VEL
LIN {X 0,Y 502.781,Z 149.86,A -85,B 0,C 180,E1 -5814.168,E2 -5814.168} C_VEL
LIN {X 0,Y 502.836,Z 149.854,A -85,B 0,C 180,E1 -5816.993,E2 -5816.993} C_VEL
LIN {X 0,Y 502.826,Z 149.907,A -85,B 0,C 180,E1 -5819.091,E2 -5819.091} C_VEL
LIN {X 0,Y 504.378,Z 157.122,A -85,B 0,C 180,E1 -5821.383,E2 -5821.383} C_VEL
LIN {X 0,Y 505.237,Z 162.472,A -85,B 0,C 180,E1 -5822.906,E2 -5822.906} C_VEL
LIN {X 0,Y 504.63,Z 172.077,A -85,B 0,C 180,E1 -5825.302,E2 -5825.302} C_VEL
LIN {X 0,Y 503.864,Z 184.95,A -85,B 0,C 180,E1 -5828.306,E2 -5828.306} C_VEL
LIN {X 0,Y 503.345,Z 198.391,A -85,B 0,C 180,E1 -5831.267,E2 -5831.267} C_VEL
LIN {X 0,Y 502.937,Z 212.128,A -85,B 0,C 180,E1 -5834.186,E2 -5834.186} C_VEL
LIN {X 0,Y 502.787,Z 220.624,A -85,B 0,C 180,E1 -5835.943,E2 -5835.943} C_VEL
LIN {X 0,Y 504.167,Z 233.243,A -85,B 0,C 180,E1 -5836.265,E2 -5836.265} C_VEL
LIN {X 0,Y 504.005,Z 246.022,A -85,B 0,C 180,E1 -5836.697,E2 -5836.697} C_VEL
LIN {X 0,Y 503.695,Z 258.11,A -85,B 0,C 180,E1 -5837.268,E2 -5837.268} C_VEL
LIN {X 0,Y 503.394,Z 270.028,A -85,B 0,C 180,E1 -5838.013,E2 -5838.013} C_VEL
LIN {X 0,Y 503.107,Z 280.336,A -85,B 0,C 180,E1 -5838.823,E2 -5838.823} C_VEL
LIN {X 0,Y 502.828,Z 289.771,A -85,B 0,C 180,E1 -5839.734,E2 -5839.734} C_VEL
LIN {X 0,Y 502.597,Z 298.325,A -85,B 0,C 180,E1 -5840.745,E2 -5840.745} C_VEL
LIN {X 0,Y 502.409,Z 306.655,A -85,B 0,C 180,E1 -5841.958,E2 -5841.958} C_VEL
LIN {X 0,Y 502.24,Z 313.341,A -85,B 0,C 180,E1 -5843.168,E2 -5843.168} C_VEL
LIN {X 0,Y 502.221,Z 318.649,A -85,B 0,C 180,E1 -5844.377,E2 -5844.377} C_VEL
LIN {X 0,Y 502.117,Z 322.746,A -85,B 0,C 180,E1 -5845.584,E2 -5845.584} C_VEL
LIN {X 0,Y 502.123,Z 325.77,A -85,B 0,C 180,E1 -5846.789,E2 -5846.789} C_VEL
LIN {X 0,Y 502.121,Z 327.218,A -85,B 0,C 180,E1 -5847.592,E2 -5847.592} C_VEL
LIN {X 0,Y 502,Z 328.873,A -85,B 0,C 180,E1 -5849.197,E2 -5849.197} C_VEL
LIN {X 0,Y 501.998,Z 329.105,A -85,B 0,C 180,E1 -5849.999,E2 -5849.999} C_VEL
LIN {X 0,Y 502.036,Z 328.283,A -85,B 0,C 180,E1 -5851.603,E2 -5851.603} C_VEL
LIN {X 0,Y 502.121,Z 327.283,A -85,B 0,C 180,E1 -5852.405,E2 -5852.405} C_VEL
LIN {X 0,Y 502.122,Z 325.854,A -85,B 0,C 180,E1 -5853.208,E2 -5853.208} C_VEL
LIN {X 0,Y 502.105,Z 322.864,A -85,B 0,C 180,E1 -5854.414,E2 -5854.414} C_VEL
LIN {X 0,Y 502.221,Z 318.806,A -85,B 0,C 180,E1 -5855.62,E2 -5855.62} C_VEL
LIN {X 0,Y 502.326,Z 312.638,A -85,B 0,C 180,E1 -5857.01,E2 -5857.01} C_VEL
LIN {X 0,Y 502.432,Z 305.687,A -85,B 0,C 180,E1 -5858.242,E2 -5858.242} C_VEL
LIN {X 0,Y 502.616,Z 298.681,A -85,B 0,C 180,E1 -5859.252,E2 -5859.252} C_VEL
LIN {X 0,Y 502.844,Z 290.221,A -85,B 0,C 180,E1 -5860.264,E2 -5860.264} C_VEL
LIN {X 0,Y 503.215,Z 279.736,A -85,B 0,C 180,E1 -5861.274,E2 -5861.274} C_VEL
LIN {X 0,Y 503.485,Z 267.883,A -85,B 0,C 180,E1 -5862.188,E2 -5862.188} C_VEL
LIN {X 0,Y 503.806,Z 255.938,A -85,B 0,C 180,E1 -5862.895,E2 -5862.895} C_VEL
LIN {X 0,Y 504.106,Z 243.494,A -85,B 0,C 180,E1 -5863.452,E2 -5863.452} C_VEL
LIN {X 0,Y 504.163,Z 231.53,A -85,B 0,C 180,E1 -5863.835,E2 -5863.835} C_VEL
LIN {X 0,Y 502.799,Z 220.691,A -85,B 0,C 180,E1 -5864.106,E2 -5864.106} C_VEL
LIN {X 0,Y 503.178,Z 204.579,A -85,B 0,C 180,E1 -5867.474,E2 -5867.474} C_VEL
LIN {X 0,Y 503.659,Z 190.699,A -85,B 0,C 180,E1 -5870.415,E2 -5870.415} C_VEL
LIN {X 0,Y 504.164,Z 176.933,A -85,B 0,C 180,E1 -5873.407,E2 -5873.407} C_VEL
LIN {X 0,Y 504.803,Z 163.246,A -85,B 0,C 180,E1 -5876.454,E2 -5876.454} C_VEL
LIN {X 0,Y 504.692,Z 159.333,A -85,B 0,C 180,E1 -5877.355,E2 -5877.355} C_VEL
LIN {X 0,Y 502.827,Z 149.853,A -85,B 0,C 180,E1 -5879.695,E2 -5879.695} C_VEL
LIN {X 0,Y 502.826,Z 149.851,A -85,B 0,C 180,E1 -5883.03,E2 -5883.03} C_VEL
LIN {X 0,Y 502.778,Z 149.861,A -85,B 0,C 180,E1 -5885.949,E2 -5885.949} C_VEL
LIN {X 0,Y 502.791,Z 149.858,A -85,B 0,C 180,E1 -5888.975,E2 -5888.975} C_VEL
LIN {X 0,Y 502.794,Z 149.855,A -85,B 0,C 180,E1 -5892.198,E2 -5892.198} C_VEL
LIN {X 0,Y 502.792,Z 149.856,A -85,B 0,C 180,E1 -5895.467,E2 -5895.467} C_VEL
LIN {X 0,Y 502.82,Z 149.853,A -85,B 0,C 180,E1 -5897.863,E2 -5897.863} C_VEL
LIN {X 0,Y 502.811,Z 149.854,A -85,B 0,C 180,E1 -5901.025,E2 -5901.025} C_VEL
LIN {X 0,Y 502.758,Z 149.863,A -85,B 0,C 180,E1 -5904.169,E2 -5904.169} C_VEL
LIN {X 0,Y 502.821,Z 149.85,A -85,B 0,C 180,E1 -5906.992,E2 -5906.992} C_VEL
LIN {X 0,Y 502.818,Z 149.851,A -85,B 0,C 180,E1 -5910.061,E2 -5910.061} C_VEL
LIN {X 0,Y 502.823,Z 149.854,A -85,B 0,C 180,E1 -5912.532,E2 -5912.532} C_VEL
LIN {X 0,Y 502.809,Z 149.851,A -85,B 0,C 180,E1 -5915.299,E2 -5915.299} C_VEL
LIN {X 0,Y 502.765,Z 149.86,A -85,B 0,C 180,E1 -5917.826,E2 -5917.826} C_VEL
LIN {X 0,Y 502.812,Z 149.851,A -85,B 0,C 180,E1 -5920.4,E2 -5920.4} C_VEL
LIN {X 0,Y 502.823,Z 149.854,A -85,B 0,C 180,E1 -5922.931,E2 -5922.931} C_VEL
LIN {X 0,Y 502.832,Z 149.849,A -85,B 0,C 180,E1 -5925.429,E2 -5925.429} C_VEL
LIN {X 0,Y 502.874,Z 149.843,A -85,B 0,C 180,E1 -5928.717,E2 -5928.717} C_VEL
LIN {X 0,Y 502.884,Z 149.842,A -85,B 0,C 180,E1 -5931.966,E2 -5931.966} C_VEL
LIN {X 0,Y 502.933,Z 149.839,A -85,B 0,C 180,E1 -5934.386,E2 -5934.386} C_VEL
LIN {X 0,Y 503.012,Z 149.83,A -85,B 0,C 180,E1 -5937.598,E2 -5937.598} C_VEL
LIN {X 0,Y 503.008,Z 149.827,A -85,B 0,C 180,E1 -5940,E2 -5940} C_VEL
LIN {X 0,Y 503.002,Z 149.828,A -85,B 0,C 180,E1 -5942.402,E2 -5942.402} C_VEL
LIN {X 0,Y 502.924,Z 149.838,A -85,B 0,C 180,E1 -5945.614,E2 -5945.614} C_VEL
LIN {X 0,Y 502.888,Z 149.846,A -85,B 0,C 180,E1 -5948.034,E2 -5948.034} C_VEL
LIN {X 0,Y 502.881,Z 149.846,A -85,B 0,C 180,E1 -5951.283,E2 -5951.283} C_VEL
LIN {X 0,Y 502.835,Z 149.854,A -85,B 0,C 180,E1 -5954.571,E2 -5954.571} C_VEL
LIN {X 0,Y 502.847,Z 149.85,A -85,B 0,C 180,E1 -5957.907,E2 -5957.907} C_VEL
LIN {X 0,Y 502.816,Z 149.851,A -85,B 0,C 180,E1 -5960.537,E2 -5960.537} C_VEL
LIN {X 0,Y 502.792,Z 149.857,A -85,B 0,C 180,E1 -5963.041,E2 -5963.041} C_VEL
LIN {X 0,Y 502.792,Z 149.853,A -85,B 0,C 180,E1 -5965.678,E2 -5965.678} C_VEL
LIN {X 0,Y 502.782,Z 149.856,A -85,B 0,C 180,E1 -5968.376,E2 -5968.376} C_VEL
LIN {X 0,Y 502.786,Z 149.857,A -85,B 0,C 180,E1 -5971.144,E2 -5971.144} C_VEL
LIN {X 0,Y 502.797,Z 149.854,A -85,B 0,C 180,E1 -5973.994,E2 -5973.994} C_VEL
LIN {X 0,Y 502.769,Z 149.856,A -85,B 0,C 180,E1 -5977.179,E2 -5977.179} C_VEL
LIN {X 0,Y 502.776,Z 149.857,A -85,B 0,C 180,E1 -5980.016,E2 -5980.016} C_VEL
LIN {X 0,Y 502.792,Z 149.853,A -85,B 0,C 180,E1 -5982.2,E2 -5982.2} C_VEL
LIN {X 0,Y 502.791,Z 149.854,A -85,B 0,C 180,E1 -5985.47,E2 -5985.47} C_VEL
LIN {X 0,Y 502.821,Z 149.853,A -85,B 0,C 180,E1 -5987.866,E2 -5987.866} C_VEL
LIN {X 0,Y 502.792,Z 149.854,A -85,B 0,C 180,E1 -5991.025,E2 -5991.025} C_VEL
LIN {X 0,Y 502.763,Z 149.856,A -85,B 0,C 180,E1 -5994.171,E2 -5994.171} C_VEL
LIN {X 0,Y 502.802,Z 149.853,A -85,B 0,C 180,E1 -5997.245,E2 -5997.245} C_VEL
LIN {X 0,Y 502.105,Z 149.942,A -85,B 0,C 180,E1 -5997.913,E2 -5997.913} C_VEL
LIN {X 0,Y 499.247,Z 150.296,A -85,B 0,C 180,E1 -5998.999,E2 -5998.999} C_VEL
LIN {X 0,Y 496.855,Z 150.596,A -85,B 0,C 180,E1 -5999.874,E2 -5999.874} C_VEL
LIN {X 0,Y 495.838,Z 150.721,A -85,B 0,C 180,E1 -6000.55,E2 -6000.55} C_VEL
LIN {X 0,Y 495.759,Z 150.73,A -85,B 0,C 180,E1 -6000.779,E2 -6000.779} C_VEL
LIN {X 0,Y 495.801,Z 150.729,A -85,B 0,C 180,E1 -6003.256,E2 -6003.256} C_VEL
LIN {X 0,Y 495.734,Z 150.738,A -85,B 0,C 180,E1 -6006.614,E2 -6006.614} C_VEL
LIN {X 0,Y 495.775,Z 150.728,A -85,B 0,C 180,E1 -6009.326,E2 -6009.326} C_VEL
LIN {X 0,Y 495.796,Z 150.729,A -85,B 0,C 180,E1 -6011.831,E2 -6011.831} C_VEL
LIN {X 0,Y 495.822,Z 150.723,A -85,B 0,C 180,E1 -6014.55,E2 -6014.55} C_VEL
LIN {X 0,Y 495.828,Z 150.722,A -85,B 0,C 180,E1 -6017.967,E2 -6017.967} C_VEL
LIN {X 0,Y 495.837,Z 150.72,A -85,B 0,C 180,E1 -6021.032,E2 -6021.032} C_VEL
LIN {X 0,Y 495.881,Z 150.718,A -85,B 0,C 180,E1 -6023.491,E2 -6023.491} C_VEL
LIN {X 0,Y 495.843,Z 150.723,A -85,B 0,C 180,E1 -6026.751,E2 -6026.751} C_VEL
LIN {X 0,Y 495.87,Z 150.721,A -85,B 0,C 180,E1 -6028.377,E2 -6028.377} C_VEL
LIN {X 0,Y 495.974,Z 150.707,A -85,B 0,C 180,E1 -6030.001,E2 -6030.001} C_VEL
LIN {X 0,Y 495.988,Z 150.701,A -85,B 0,C 180,E1 -6032.438,E2 -6032.438} C_VEL
LIN {X 0,Y 495.897,Z 150.714,A -85,B 0,C 180,E1 -6035.695,E2 -6035.695} C_VEL
LIN {X 0,Y 495.875,Z 150.718,A -85,B 0,C 180,E1 -6038.149,E2 -6038.149} C_VEL
LIN {X 0,Y 495.855,Z 150.719,A -85,B 0,C 180,E1 -6041.446,E2 -6041.446} C_VEL
LIN {X 0,Y 495.779,Z 150.728,A -85,B 0,C 180,E1 -6044.784,E2 -6044.784} C_VEL
LIN {X 0,Y 495.768,Z 150.731,A -85,B 0,C 180,E1 -6047.32,E2 -6047.32} C_VEL
LIN {X 0,Y 495.776,Z 150.73,A -85,B 0,C 180,E1 -6049.891,E2 -6049.891} C_VEL
LIN {X 0,Y 495.762,Z 150.729,A -85,B 0,C 180,E1 -6052.861,E2 -6052.861} C_VEL
LIN {X 0,Y 495.72,Z 150.733,A -85,B 0,C 180,E1 -6056.073,E2 -6056.073} C_VEL
LIN {X 0,Y 495.733,Z 150.737,A -85,B 0,C 180,E1 -6058.818,E2 -6058.818} C_VEL
LIN {X 0,Y 495.759,Z 150.733,A -85,B 0,C 180,E1 -6061.726,E2 -6061.726} C_VEL
LIN {X 0,Y 495.766,Z 150.729,A -85,B 0,C 180,E1 -6064.693,E2 -6064.693} C_VEL
LIN {X 0,Y 495.709,Z 150.736,A -85,B 0,C 180,E1 -6067.565,E2 -6067.565} C_VEL
LIN {X 0,Y 495.735,Z 150.735,A -85,B 0,C 180,E1 -6070.704,E2 -6070.704} C_VEL
LIN {X 0,Y 495.729,Z 150.737,A -85,B 0,C 180,E1 -6074.003,E2 -6074.003} C_VEL
LIN {X 0,Y 495.73,Z 150.737,A -85,B 0,C 180,E1 -6077.117,E2 -6077.117} C_VEL
LIN {X 0,Y 495.759,Z 150.73,A -85,B 0,C 180,E1 -6079.954,E2 -6079.954} C_VEL
LIN {X 0,Y 495.711,Z 150.737,A -85,B 0,C 180,E1 -6082.557,E2 -6082.557} C_VEL
LIN {X 0,Y 495.774,Z 150.732,A -85,B 0,C 180,E1 -6085.456,E2 -6085.456} C_VEL
LIN {X 0,Y 495.817,Z 150.829,A -85,B 0,C 180,E1 -6088.487,E2 -6088.487} C_VEL
LIN {X 0,Y 496.36,Z 155.524,A -85,B 0,C 180,E1 -6090.293,E2 -6090.293} C_VEL
LIN {X 0,Y 496.159,Z 163.298,A -85,B 0,C 180,E1 -6093.176,E2 -6093.176} C_VEL
LIN {X 0,Y 495.905,Z 171.54,A -85,B 0,C 180,E1 -6096.178,E2 -6096.178} C_VEL
LIN {X 0,Y 495.731,Z 180.329,A -85,B 0,C 180,E1 -6099.341,E2 -6099.341} C_VEL
LIN {X 0,Y 495.538,Z 189.763,A -85,B 0,C 180,E1 -6102.672,E2 -6102.672} C_VEL
LIN {X 0,Y 495.401,Z 198.206,A -85,B 0,C 180,E1 -6105.625,E2 -6105.625} C_VEL
LIN {X 0,Y 495.292,Z 206.646,A -85,B 0,C 180,E1 -6108.542,E2 -6108.542} C_VEL
LIN {X 0,Y 495.156,Z 214.782,A -85,B 0,C 180,E1 -6111.326,E2 -6111.326} C_VEL
LIN {X 0,Y 496.187,Z 224.688,A -85,B 0,C 180,E1 -6111.755,E2 -6111.755} C_VEL
LIN {X 0,Y 495.977,Z 233.736,A -85,B 0,C 180,E1 -6112.264,E2 -6112.264} C_VEL
LIN {X 0,Y 495.754,Z 242.331,A -85,B 0,C 180,E1 -6112.911,E2 -6112.911} C_VEL
LIN {X 0,Y 495.541,Z 250.251,A -85,B 0,C 180,E1 -6113.69,E2 -6113.69} C_VEL
LIN {X 0,Y 495.45,Z 256.717,A -85,B 0,C 180,E1 -6114.506,E2 -6114.506} C_VEL
LIN {X 0,Y 495.321,Z 262.911,A -85,B 0,C 180,E1 -6115.524,E2 -6115.524} C_VEL
LIN {X 0,Y 495.256,Z 268.256,A -85,B 0,C 180,E1 -6116.746,E2 -6116.746} C_VEL
LIN {X 0,Y 495.085,Z 270.791,A -85,B 0,C 180,E1 -6117.559,E2 -6117.559} C_VEL
LIN {X 0,Y 494.981,Z 272.577,A -85,B 0,C 180,E1 -6118.373,E2 -6118.373} C_VEL
LIN {X 0,Y 494.942,Z 273.661,A -85,B 0,C 180,E1 -6119.186,E2 -6119.186} C_VEL
LIN {X 0,Y 494.935,Z 274.072,A -85,B 0,C 180,E1 -6120,E2 -6120} C_VEL
LIN {X 0,Y 494.944,Z 273.816,A -85,B 0,C 180,E1 -6120.814,E2 -6120.814} C_VEL
LIN {X 0,Y 494.984,Z 272.889,A -85,B 0,C 180,E1 -6121.627,E2 -6121.627} C_VEL
LIN {X 0,Y 495.141,Z 270.187,A -85,B 0,C 180,E1 -6122.848,E2 -6122.848} C_VEL
LIN {X 0,Y 495.302,Z 267.432,A -85,B 0,C 180,E1 -6123.661,E2 -6123.661} C_VEL
LIN {X 0,Y 495.38,Z 262.803,A -85,B 0,C 180,E1 -6124.679,E2 -6124.679} C_VEL
LIN {X 0,Y 495.423,Z 256.563,A -85,B 0,C 180,E1 -6125.699,E2 -6125.699} C_VEL
LIN {X 0,Y 495.614,Z 250.075,A -85,B 0,C 180,E1 -6126.514,E2 -6126.514} C_VEL
LIN {X 0,Y 495.842,Z 241.689,A -85,B 0,C 180,E1 -6127.329,E2 -6127.329} C_VEL
LIN {X 0,Y 496.128,Z 233.492,A -85,B 0,C 180,E1 -6127.939,E2 -6127.939} C_VEL
LIN {X 0,Y 496.216,Z 223.408,A -85,B 0,C 180,E1 -6128.501,E2 -6128.501} C_VEL
LIN {X 0,Y 495.234,Z 215.19,A -85,B 0,C 180,E1 -6128.878,E2 -6128.878} C_VEL
LIN {X 0,Y 495.351,Z 206.849,A -85,B 0,C 180,E1 -6131.77,E2 -6131.77} C_VEL
LIN {X 0,Y 495.553,Z 196.656,A -85,B 0,C 180,E1 -6135.335,E2 -6135.335} C_VEL
LIN {X 0,Y 495.741,Z 187.598,A -85,B 0,C 180,E1 -6138.558,E2 -6138.558} C_VEL
LIN {X 0,Y 495.914,Z 179.163,A -85,B 0,C 180,E1 -6141.621,E2 -6141.621} C_VEL
LIN {X 0,Y 496.117,Z 172.05,A -85,B 0,C 180,E1 -6144.256,E2 -6144.256} C_VEL
LIN {X 0,Y 496.473,Z 163.843,A -85,B 0,C 180,E1 -6147.391,E2 -6147.391} C_VEL
LIN {X 0,Y 496.769,Z 157.979,A -85,B 0,C 180,E1 -6149.68,E2 -6149.68} C_VEL
LIN {X 0,Y 496.491,Z 154.558,A -85,B 0,C 180,E1 -6151.109,E2 -6151.109} C_VEL
LIN {X 0,Y 495.791,Z 150.731,A -85,B 0,C 180,E1 -6152.863,E2 -6152.863} C_VEL
LIN {X 0,Y 495.753,Z 150.736,A -85,B 0,C 180,E1 -6155.538,E2 -6155.538} C_VEL
LIN {X 0,Y 495.769,Z 150.733,A -85,B 0,C 180,E1 -6158.768,E2 -6158.768} C_VEL
LIN {X 0,Y 495.762,Z 150.733,A -85,B 0,C 180,E1 -6161.781,E2 -6161.781} C_VEL
LIN {X 0,Y 495.743,Z 150.736,A -85,B 0,C 180,E1 -6165.14,E2 -6165.14} C_VEL
LIN {X 0,Y 495.762,Z 150.733,A -85,B 0,C 180,E1 -6168.218,E2 -6168.218} C_VEL
LIN {X 0,Y 495.755,Z 150.735,A -85,B 0,C 180,E1 -6171.408,E2 -6171.408} C_VEL
LIN {X 0,Y 495.753,Z 150.735,A -85,B 0,C 180,E1 -6174.462,E2 -6174.462} C_VEL
LIN {X 0,Y 495.772,Z 150.734,A -85,B 0,C 180,E1 -6177.405,E2 -6177.405} C_VEL
LIN {X 0,Y 495.785,Z 150.801,A -85,B 0,C 180,E1 -6178.603,E2 -6178.603} C_VEL
LIN {X 0,Y 497.531,Z 158.935,A -85,B 0,C 180,E1 -6181.296,E2 -6181.296} C_VEL
LIN {X 0,Y 498.356,Z 163.632,A -85,B 0,C 180,E1 -6182.679,E2 -6182.679} C_VEL
LIN {X 0,Y 497.892,Z 171.081,A -85,B 0,C 180,E1 -6184.608,E2 -6184.608} C_VEL
LIN {X 0,Y 497.063,Z 183.206,A -85,B 0,C 180,E1 -6187.557,E2 -6187.557} C_VEL
LIN {X 0,Y 496.433,Z 196.402,A -85,B 0,C 180,E1 -6190.567,E2 -6190.567} C_VEL
LIN {X 0,Y 496,Z 208.061,A -85,B 0,C 180,E1 -6193.113,E2 -6193.113} C_VEL
LIN {X 0,Y 495.73,Z 220.657,A -85,B 0,C 180,E1 -6195.791,E2 -6195.791} C_VEL
LIN {X 0,Y 497.173,Z 234.424,A -85,B 0,C 180,E1 -6196.146,E2 -6196.146} C_VEL
LIN {X 0,Y 496.982,Z 247.388,A -85,B 0,C 180,E1 -6196.61,E2 -6196.61} C_VEL
LIN {X 0,Y 496.638,Z 260.177,A -85,B 0,C 180,E1 -6197.256,E2 -6197.256} C_VEL
LIN {X 0,Y 496.354,Z 270.701,A -85,B 0,C 180,E1 -6197.944,E2 -6197.944} C_VEL
LIN {X 0,Y 496.07,Z 280.835,A -85,B 0,C 180,E1 -6198.766,E2 -6198.766} C_VEL
LIN {X 0,Y 495.723,Z 290.992,A -85,B 0,C 180,E1 -6199.791,E2 -6199.791} C_VEL
LIN {X 0,Y 495.488,Z 299.284,A -85,B 0,C 180,E1 -6200.817,E2 -6200.817} C_VEL
LIN {X 0,Y 495.318,Z 307.397,A -85,B 0,C 180,E1 -6202.047,E2 -6202.047} C_VEL
LIN {X 0,Y 495.17,Z 312.863,A -85,B 0,C 180,E1 -6203.07,E2 -6203.07} C_VEL
LIN {X 0,Y 495.134,Z 318.201,A -85,B 0,C 180,E1 -6204.297,E2 -6204.297} C_VEL
LIN {X 0,Y 495.02,Z 322.32,A -85,B 0,C 180,E1 -6205.52,E2 -6205.52} C_VEL
LIN {X 0,Y 495.046,Z 325.361,A -85,B 0,C 180,E1 -6206.743,E2 -6206.743} C_VEL
LIN {X 0,Y 495.054,Z 326.82,A -85,B 0,C 180,E1 -6207.558,E2 -6207.558} C_VEL
LIN {X 0,Y 494.919,Z 328.484,A -85,B 0,C 180,E1 -6209.185,E2 -6209.185} C_VEL
LIN {X 0,Y 494.915,Z 328.719,A -85,B 0,C 180,E1 -6209.999,E2 -6209.999} C_VEL
LIN {X 0,Y 494.963,Z 327.898,A -85,B 0,C 180,E1 -6211.626,E2 -6211.626} C_VEL
LIN {X 0,Y 495.054,Z 326.897,A -85,B 0,C 180,E1 -6212.44,E2 -6212.44} C_VEL
LIN {X 0,Y 495.045,Z 325.46,A -85,B 0,C 180,E1 -6213.254,E2 -6213.254} C_VEL
LIN {X 0,Y 495.01,Z 322.46,A -85,B 0,C 180,E1 -6214.477,E2 -6214.477} C_VEL
LIN {X 0,Y 495.134,Z 318.388,A -85,B 0,C 180,E1 -6215.701,E2 -6215.701} C_VEL
LIN {X 0,Y 495.251,Z 312.1,A -85,B 0,C 180,E1 -6217.131,E2 -6217.131} C_VEL
LIN {X 0,Y 495.357,Z 305.225,A -85,B 0,C 180,E1 -6218.36,E2 -6218.36} C_VEL
LIN {X 0,Y 495.567,Z 298.189,A -85,B 0,C 180,E1 -6219.385,E2 -6219.385} C_VEL
LIN {X 0,Y 495.817,Z 289.678,A -85,B 0,C 180,E1 -6220.411,E2 -6220.411} C_VEL
LIN {X 0,Y 496.226,Z 279.128,A -85,B 0,C 180,E1 -6221.435,E2 -6221.435} C_VEL
LIN {X 0,Y 496.442,Z 268.644,A -85,B 0,C 180,E1 -6222.259,E2 -6222.259} C_VEL
LIN {X 0,Y 496.791,Z 257.265,A -85,B 0,C 180,E1 -6222.966,E2 -6222.966} C_VEL
LIN {X 0,Y 497.137,Z 245.034,A -85,B 0,C 180,E1 -6223.54,E2 -6223.54} C_VEL
LIN {X 0,Y 497.214,Z 232.422,A -85,B 0,C 180,E1 -6223.967,E2 -6223.967} C_VEL
LIN {X 0,Y 495.712,Z 220.705,A -85,B 0,C 180,E1 -6224.259,E2 -6224.259} C_VEL
LIN {X 0,Y 496.081,Z 206.354,A -85,B 0,C 180,E1 -6227.306,E2 -6227.306} C_VEL
LIN {X 0,Y 496.614,Z 192.584,A -85,B 0,C 180,E1 -6230.285,E2 -6230.285} C_VEL
LIN {X 0,Y 497.175,Z 178.836,A -85,B 0,C 180,E1 -6233.314,E2 -6233.314} C_VEL
LIN {X 0,Y 497.835,Z 165.154,A -85,B 0,C 180,E1 -6236.402,E2 -6236.402} C_VEL
LIN {X 0,Y 497.749,Z 160.725,A -85,B 0,C 180,E1 -6237.435,E2 -6237.435} C_VEL
LIN {X 0,Y 495.773,Z 150.732,A -85,B 0,C 180,E1 -6239.961,E2 -6239.961} C_VEL
LIN {X 0,Y 495.788,Z 150.727,A -85,B 0,C 180,E1 -6243.243,E2 -6243.243} C_VEL
LIN {X 0,Y 495.723,Z 150.737,A -85,B 0,C 180,E1 -6246.089,E2 -6246.089} C_VEL
LIN {X 0,Y 495.754,Z 150.733,A -85,B 0,C 180,E1 -6248.767,E2 -6248.767} C_VEL
LIN {X 0,Y 495.74,Z 150.731,A -85,B 0,C 180,E1 -6251.78,E2 -6251.78} C_VEL
LIN {X 0,Y 495.74,Z 150.732,A -85,B 0,C 180,E1 -6255.138,E2 -6255.138} C_VEL
LIN {X 0,Y 495.769,Z 150.729,A -85,B 0,C 180,E1 -6258.22,E2 -6258.22} C_VEL
LIN {X 0,Y 495.767,Z 150.731,A -85,B 0,C 180,E1 -6261.228,E2 -6261.228} C_VEL
LIN {X 0,Y 495.732,Z 150.735,A -85,B 0,C 180,E1 -6264.461,E2 -6264.461} C_VEL
LIN {X 0,Y 495.757,Z 150.732,A -85,B 0,C 180,E1 -6267.405,E2 -6267.405} C_VEL
LIN {X 0,Y 495.769,Z 150.729,A -85,B 0,C 180,E1 -6270.254,E2 -6270.254} C_VEL
LIN {X 0,Y 495.821,Z 150.723,A -85,B 0,C 180,E1 -6273.247,E2 -6273.247} C_VEL
LIN {X 0,Y 495.728,Z 150.736,A -85,B 0,C 180,E1 -6275.724,E2 -6275.724} C_VEL
LIN {X 0,Y 495.728,Z 150.733,A -85,B 0,C 180,E1 -6278.37,E2 -6278.37} C_VEL
LIN {X 0,Y 495.771,Z 150.731,A -85,B 0,C 180,E1 -6280.971,E2 -6280.971} C_VEL
LIN {X 0,Y 495.768,Z 150.729,A -85,B 0,C 180,E1 -6283.529,E2 -6283.529} C_VEL
LIN {X 0,Y 495.781,Z 150.731,A -85,B 0,C 180,E1 -6286.055,E2 -6286.055} C_VEL
LIN {X 0,Y 495.856,Z 150.717,A -85,B 0,C 180,E1 -6288.555,E2 -6288.555} C_VEL
LIN {X 0,Y 495.856,Z 150.717,A -85,B 0,C 180,E1 -6291.852,E2 -6291.852} C_VEL
LIN {X 0,Y 495.89,Z 150.716,A -85,B 0,C 180,E1 -6294.306,E2 -6294.306} C_VEL
LIN {X 0,Y 495.981,Z 150.706,A -85,B 0,C 180,E1 -6297.564,E2 -6297.564} C_VEL
LIN {X 0,Y 495.979,Z 150.703,A -85,B 0,C 180,E1 -6300,E2 -6300} C_VEL
LIN {X 0,Y 495.971,Z 150.704,A -85,B 0,C 180,E1 -6302.436,E2 -6302.436} C_VEL
LIN {X 0,Y 495.881,Z 150.715,A -85,B 0,C 180,E1 -6305.694,E2 -6305.694} C_VEL
LIN {X 0,Y 495.859,Z 150.721,A -85,B 0,C 180,E1 -6308.148,E2 -6308.148} C_VEL
LIN {X 0,Y 495.855,Z 150.72,A -85,B 0,C 180,E1 -6311.445,E2 -6311.445} C_VEL
LIN {X 0,Y 495.778,Z 150.73,A -85,B 0,C 180,E1 -6314.783,E2 -6314.783} C_VEL
LIN {X 0,Y 495.773,Z 150.728,A -85,B 0,C 180,E1 -6317.319,E2 -6317.319} C_VEL
LIN {X 0,Y 495.764,Z 150.733,A -85,B 0,C 180,E1 -6319.891,E2 -6319.891} C_VEL
LIN {X 0,Y 495.751,Z 150.735,A -85,B 0,C 180,E1 -6322.863,E2 -6322.863} C_VEL
LIN {X 0,Y 495.75,Z 150.734,A -85,B 0,C 180,E1 -6326.07,E2 -6326.07} C_VEL
LIN {X 0,Y 495.731,Z 150.732,A -85,B 0,C 180,E1 -6328.817,E2 -6328.817} C_VEL
LIN {X 0,Y 495.747,Z 150.734,A -85,B 0,C 180,E1 -6331.727,E2 -6331.727} C_VEL
LIN {X 0,Y 495.766,Z 150.732,A -85,B 0,C 180,E1 -6334.697,E2 -6334.697} C_VEL
LIN {X 0,Y 495.719,Z 150.736,A -85,B 0,C 180,E1 -6337.563,E2 -6337.563} C_VEL
LIN {X 0,Y 495.755,Z 150.729,A -85,B 0,C 180,E1 -6340.701,E2 -6340.701} C_VEL
LIN {X 0,Y 495.724,Z 150.734,A -85,B 0,C 180,E1 -6344.002,E2 -6344.002} C_VEL
LIN {X 0,Y 495.725,Z 150.735,A -85,B 0,C 180,E1 -6347.119,E2 -6347.119} C_VEL
LIN {X 0,Y 495.75,Z 150.734,A -85,B 0,C 180,E1 -6349.954,E2 -6349.954} C_VEL
LIN {X 0,Y 495.717,Z 150.734,A -85,B 0,C 180,E1 -6352.555,E2 -6352.555} C_VEL
LIN {X 0,Y 495.77,Z 150.729,A -85,B 0,C 180,E1 -6355.458,E2 -6355.458} C_VEL
LIN {X 0,Y 495.754,Z 150.734,A -85,B 0,C 180,E1 -6358.366,E2 -6358.366} C_VEL
LIN {X 0,Y 495.759,Z 150.73,A -85,B 0,C 180,E1 -6360.779,E2 -6360.779} C_VEL
LIN {X 0,Y 495.096,Z 150.817,A -85,B 0,C 180,E1 -6361.457,E2 -6361.457} C_VEL
LIN {X 0,Y 492.226,Z 151.17,A -85,B 0,C 180,E1 -6362.559,E2 -6362.559} C_VEL
LIN {X 0,Y 489.804,Z 151.474,A -85,B 0,C 180,E1 -6363.447,E2 -6363.447} C_VEL
LIN {X 0,Y 488.777,Z 151.599,A -85,B 0,C 180,E1 -6364.133,E2 -6364.133} C_VEL
LIN {X 0,Y 488.701,Z 151.609,A -85,B 0,C 180,E1 -6364.366,E2 -6364.366} C_VEL
LIN {X 0,Y 488.716,Z 151.607,A -85,B 0,C 180,E1 -6367.155,E2 -6367.155} C_VEL
LIN {X 0,Y 488.723,Z 151.609,A -85,B 0,C 180,E1 -6369.812,E2 -6369.812} C_VEL
LIN {X 0,Y 488.732,Z 151.606,A -85,B 0,C 180,E1 -6372.425,E2 -6372.425} C_VEL
LIN {X 0,Y 488.758,Z 151.605,A -85,B 0,C 180,E1 -6375.001,E2 -6375.001} C_VEL
LIN {X 0,Y 488.804,Z 151.601,A -85,B 0,C 180,E1 -6378.389,E2 -6378.389} C_VEL
LIN {X 0,Y 488.816,Z 151.598,A -85,B 0,C 180,E1 -6381.735,E2 -6381.735} C_VEL
LIN {X 0,Y 488.856,Z 151.59,A -85,B 0,C 180,E1 -6384.226,E2 -6384.226} C_VEL
LIN {X 0,Y 488.962,Z 151.577,A -85,B 0,C 180,E1 -6387.53,E2 -6387.53} C_VEL
LIN {X 0,Y 488.943,Z 151.583,A -85,B 0,C 180,E1 -6390.001,E2 -6390.001} C_VEL
LIN {X 0,Y 488.955,Z 151.577,A -85,B 0,C 180,E1 -6392.473,E2 -6392.473} C_VEL
LIN {X 0,Y 488.857,Z 151.591,A -85,B 0,C 180,E1 -6395.777,E2 -6395.777} C_VEL
LIN {X 0,Y 488.819,Z 151.598,A -85,B 0,C 180,E1 -6398.268,E2 -6398.268} C_VEL
LIN {X 0,Y 488.809,Z 151.598,A -85,B 0,C 180,E1 -6401.614,E2 -6401.614} C_VEL
LIN {X 0,Y 488.757,Z 151.604,A -85,B 0,C 180,E1 -6405.002,E2 -6405.002} C_VEL
LIN {X 0,Y 488.751,Z 151.605,A -85,B 0,C 180,E1 -6408.443,E2 -6408.443} C_VEL
LIN {X 0,Y 488.712,Z 151.608,A -85,B 0,C 180,E1 -6411.072,E2 -6411.072} C_VEL
LIN {X 0,Y 488.673,Z 151.615,A -85,B 0,C 180,E1 -6413.748,E2 -6413.748} C_VEL
LIN {X 0,Y 488.702,Z 151.613,A -85,B 0,C 180,E1 -6416.922,E2 -6416.922} C_VEL
LIN {X 0,Y 488.723,Z 151.609,A -85,B 0,C 180,E1 -6420.22,E2 -6420.22} C_VEL
LIN {X 0,Y 488.734,Z 151.609,A -85,B 0,C 180,E1 -6423.484,E2 -6423.484} C_VEL
LIN {X 0,Y 488.672,Z 151.613,A -85,B 0,C 180,E1 -6426.353,E2 -6426.353} C_VEL
LIN {X 0,Y 488.688,Z 151.61,A -85,B 0,C 180,E1 -6429.257,E2 -6429.257} C_VEL
LIN {X 0,Y 488.675,Z 151.614,A -85,B 0,C 180,E1 -6432.528,E2 -6432.528} C_VEL
LIN {X 0,Y 488.706,Z 151.612,A -85,B 0,C 180,E1 -6435.198,E2 -6435.198} C_VEL
LIN {X 0,Y 488.712,Z 151.611,A -85,B 0,C 180,E1 -6438.585,E2 -6438.585} C_VEL
LIN {X 0,Y 488.694,Z 151.609,A -85,B 0,C 180,E1 -6440.95,E2 -6440.95} C_VEL
LIN {X 0,Y 488.67,Z 151.617,A -85,B 0,C 180,E1 -6443.867,E2 -6443.867} C_VEL
LIN {X 0,Y 488.742,Z 151.607,A -85,B 0,C 180,E1 -6446.877,E2 -6446.877} C_VEL
LIN {X 0,Y 488.759,Z 151.648,A -85,B 0,C 180,E1 -6448.342,E2 -6448.342} C_VEL
LIN {X 0,Y 489.313,Z 155.413,A -85,B 0,C 180,E1 -6449.821,E2 -6449.821} C_VEL
LIN {X 0,Y 489.201,Z 161.636,A -85,B 0,C 180,E1 -6452.166,E2 -6452.166} C_VEL
LIN {X 0,Y 488.933,Z 170.269,A -85,B 0,C 180,E1 -6455.364,E2 -6455.364} C_VEL
LIN {X 0,Y 488.726,Z 178.848,A -85,B 0,C 180,E1 -6458.488,E2 -6458.488} C_VEL
LIN {X 0,Y 488.533,Z 187.349,A -85,B 0,C 180,E1 -6461.549,E2 -6461.549} C_VEL
LIN {X 0,Y 488.426,Z 195.949,A -85,B 0,C 180,E1 -6464.596,E2 -6464.596} C_VEL
LIN {X 0,Y 488.247,Z 206.21,A -85,B 0,C 180,E1 -6468.188,E2 -6468.188} C_VEL
LIN {X 0,Y 488.102,Z 214.823,A -85,B 0,C 180,E1 -6471.174,E2 -6471.174} C_VEL
LIN {X 0,Y 489.178,Z 225.201,A -85,B 0,C 180,E1 -6471.636,E2 -6471.636} C_VEL
LIN {X 0,Y 488.95,Z 235.669,A -85,B 0,C 180,E1 -6472.256,E2 -6472.256} C_VEL
LIN {X 0,Y 488.669,Z 244.891,A -85,B 0,C 180,E1 -6473.009,E2 -6473.009} C_VEL
LIN {X 0,Y 488.443,Z 252.361,A -85,B 0,C 180,E1 -6473.805,E2 -6473.805} C_VEL
LIN {X 0,Y 488.417,Z 258.434,A -85,B 0,C 180,E1 -6474.633,E2 -6474.633} C_VEL
LIN {X 0,Y 488.228,Z 264.296,A -85,B 0,C 180,E1 -6475.666,E2 -6475.666} C_VEL
LIN {X 0,Y 488.175,Z 268.615,A -85,B 0,C 180,E1 -6476.699,E2 -6476.699} C_VEL
LIN {X 0,Y 488.024,Z 271.158,A -85,B 0,C 180,E1 -6477.524,E2 -6477.524} C_VEL
LIN {X 0,Y 487.91,Z 272.954,A -85,B 0,C 180,E1 -6478.349,E2 -6478.349} C_VEL
LIN {X 0,Y 487.864,Z 274.049,A -85,B 0,C 180,E1 -6479.175,E2 -6479.175} C_VEL
LIN {X 0,Y 487.854,Z 274.469,A -85,B 0,C 180,E1 -6480,E2 -6480} C_VEL
LIN {X 0,Y 487.865,Z 274.222,A -85,B 0,C 180,E1 -6480.825,E2 -6480.825} C_VEL
LIN {X 0,Y 487.913,Z 273.303,A -85,B 0,C 180,E1 -6481.651,E2 -6481.651} C_VEL
LIN {X 0,Y 488.083,Z 270.616,A -85,B 0,C 180,E1 -6482.889,E2 -6482.889} C_VEL
LIN {X 0,Y 488.249,Z 267.875,A -85,B 0,C 180,E1 -6483.714,E2 -6483.714} C_VEL
LIN {X 0,Y 488.338,Z 263.272,A -85,B 0,C 180,E1 -6484.747,E2 -6484.747} C_VEL
LIN {X 0,Y 488.386,Z 257.065,A -85,B 0,C 180,E1 -6485.781,E2 -6485.781} C_VEL
LIN {X 0,Y 488.595,Z 250.617,A -85,B 0,C 180,E1 -6486.608,E2 -6486.608} C_VEL
LIN {X 0,Y 488.831,Z 242.341,A -85,B 0,C 180,E1 -6487.435,E2 -6487.435} C_VEL
LIN {X 0,Y 489.203,Z 232.713,A -85,B 0,C 180,E1 -6488.156,E2 -6488.156} C_VEL
LIN {X 0,Y 489.188,Z 223.457,A -85,B 0,C 180,E1 -6488.676,E2 -6488.676} C_VEL
LIN {X 0,Y 488.178,Z 215.31,A -85,B 0,C 180,E1 -6489.06,E2 -6489.06} C_VEL
LIN {X 0,Y 488.284,Z 207.402,A -85,B 0,C 180,E1 -6491.832,E2 -6491.832} C_VEL
LIN {X 0,Y 488.495,Z 198.459,A -85,B 0,C 180,E1 -6495.009,E2 -6495.009} C_VEL
LIN {X 0,Y 488.7,Z 189.213,A -85,B 0,C 180,E1 -6498.349,E2 -6498.349} C_VEL
LIN {X 0,Y 488.909,Z 180.654,A -85,B 0,C 180,E1 -6501.504,E2 -6501.504} C_VEL
LIN {X 0,Y 489.159,Z 172.414,A -85,B 0,C 180,E1 -6504.624,E2 -6504.624} C_VEL
LIN {X 0,Y 489.516,Z 165.359,A -85,B 0,C 180,E1 -6507.35,E2 -6507.35} C_VEL
LIN {X 0,Y 489.846,Z 159.612,A -85,B 0,C 180,E1 -6509.669,E2 -6509.669} C_VEL
LIN {X 0,Y 489.429,Z 155.18,A -85,B 0,C 180,E1 -6511.581,E2 -6511.581} C_VEL
LIN {X 0,Y 488.763,Z 151.606,A -85,B 0,C 180,E1 -6513.301,E2 -6513.301} C_VEL
LIN {X 0,Y 488.688,Z 151.615,A -85,B 0,C 180,E1 -6516.354,E2 -6516.354} C_VEL
LIN {X 0,Y 488.707,Z 151.613,A -85,B 0,C 180,E1 -6519.254,E2 -6519.254} C_VEL
LIN {X 0,Y 488.713,Z 151.612,A -85,B 0,C 180,E1 -6521.599,E2 -6521.599} C_VEL
LIN {X 0,Y 488.707,Z 151.612,A -85,B 0,C 180,E1 -6524.802,E2 -6524.802} C_VEL
LIN {X 0,Y 488.698,Z 151.613,A -85,B 0,C 180,E1 -6527.474,E2 -6527.474} C_VEL
LIN {X 0,Y 488.739,Z 151.608,A -85,B 0,C 180,E1 -6529.676,E2 -6529.676} C_VEL
LIN {X 0,Y 488.685,Z 151.615,A -85,B 0,C 180,E1 -6532.841,E2 -6532.841} C_VEL
LIN {X 0,Y 488.73,Z 151.61,A -85,B 0,C 180,E1 -6535.886,E2 -6535.886} C_VEL
LIN {X 0,Y 488.711,Z 151.632,A -85,B 0,C 180,E1 -6538.045,E2 -6538.045} C_VEL
LIN {X 0,Y 490.175,Z 158.115,A -85,B 0,C 180,E1 -6540.352,E2 -6540.352} C_VEL
LIN {X 0,Y 491.439,Z 164.807,A -85,B 0,C 180,E1 -6542.456,E2 -6542.456} C_VEL
LIN {X 0,Y 491.292,Z 169.314,A -85,B 0,C 180,E1 -6543.674,E2 -6543.674} C_VEL
LIN {X 0,Y 490.376,Z 180.517,A -85,B 0,C 180,E1 -6546.526,E2 -6546.526} C_VEL
LIN {X 0,Y 489.568,Z 194.565,A -85,B 0,C 180,E1 -6549.846,E2 -6549.846} C_VEL
LIN {X 0,Y 489.079,Z 206.015,A -85,B 0,C 180,E1 -6552.435,E2 -6552.435} C_VEL
LIN {X 0,Y 488.65,Z 220.672,A -85,B 0,C 180,E1 -6555.621,E2 -6555.621} C_VEL
LIN {X 0,Y 490.22,Z 234.954,A -85,B 0,C 180,E1 -6555.999,E2 -6555.999} C_VEL
LIN {X 0,Y 490.006,Z 247.616,A -85,B 0,C 180,E1 -6556.468,E2 -6556.468} C_VEL
LIN {X 0,Y 489.661,Z 258.851,A -85,B 0,C 180,E1 -6557.039,E2 -6557.039} C_VEL
LIN {X 0,Y 489.34,Z 269.674,A -85,B 0,C 180,E1 -6557.746,E2 -6557.746} C_VEL
LIN {X 0,Y 489.051,Z 280.184,A -85,B 0,C 180,E1 -6558.602,E2 -6558.602} C_VEL
LIN {X 0,Y 488.69,Z 290.415,A -85,B 0,C 180,E1 -6559.643,E2 -6559.643} C_VEL
LIN {X 0,Y 488.389,Z 300.264,A -85,B 0,C 180,E1 -6560.891,E2 -6560.891} C_VEL
LIN {X 0,Y 488.2,Z 308.071,A -85,B 0,C 180,E1 -6562.138,E2 -6562.138} C_VEL
LIN {X 0,Y 488.094,Z 314.726,A -85,B 0,C 180,E1 -6563.477,E2 -6563.477} C_VEL
LIN {X 0,Y 488.044,Z 319.244,A -85,B 0,C 180,E1 -6564.628,E2 -6564.628} C_VEL
LIN {X 0,Y 487.96,Z 323.009,A -85,B 0,C 180,E1 -6565.869,E2 -6565.869} C_VEL
LIN {X 0,Y 487.971,Z 324.951,A -85,B 0,C 180,E1 -6566.696,E2 -6566.696} C_VEL
LIN {X 0,Y 487.96,Z 326.421,A -85,B 0,C 180,E1 -6567.522,E2 -6567.522} C_VEL
LIN {X 0,Y 487.893,Z 327.457,A -85,B 0,C 180,E1 -6568.348,E2 -6568.348} C_VEL
LIN {X 0,Y 487.842,Z 328.095,A -85,B 0,C 180,E1 -6569.173,E2 -6569.173} C_VEL
LIN {X 0,Y 487.835,Z 328.332,A -85,B 0,C 180,E1 -6569.999,E2 -6569.999} C_VEL
LIN {X 0,Y 487.842,Z 328.121,A -85,B 0,C 180,E1 -6570.824,E2 -6570.824} C_VEL
LIN {X 0,Y 487.893,Z 327.514,A -85,B 0,C 180,E1 -6571.65,E2 -6571.65} C_VEL
LIN {X 0,Y 487.959,Z 326.509,A -85,B 0,C 180,E1 -6572.475,E2 -6572.475} C_VEL
LIN {X 0,Y 487.969,Z 325.066,A -85,B 0,C 180,E1 -6573.301,E2 -6573.301} C_VEL
LIN {X 0,Y 487.922,Z 322.056,A -85,B 0,C 180,E1 -6574.542,E2 -6574.542} C_VEL
LIN {X 0,Y 488.027,Z 317.968,A -85,B 0,C 180,E1 -6575.784,E2 -6575.784} C_VEL
LIN {X 0,Y 488.176,Z 311.662,A -85,B 0,C 180,E1 -6577.235,E2 -6577.235} C_VEL
LIN {X 0,Y 488.304,Z 304.764,A -85,B 0,C 180,E1 -6578.482,E2 -6578.482} C_VEL
LIN {X 0,Y 488.514,Z 297.693,A -85,B 0,C 180,E1 -6579.522,E2 -6579.522} C_VEL
LIN {X 0,Y 488.798,Z 289.118,A -85,B 0,C 180,E1 -6580.562,E2 -6580.562} C_VEL
LIN {X 0,Y 489.17,Z 278.495,A -85,B 0,C 180,E1 -6581.602,E2 -6581.602} C_VEL
LIN {X 0,Y 489.469,Z 267.346,A -85,B 0,C 180,E1 -6582.479,E2 -6582.479} C_VEL
LIN {X 0,Y 489.852,Z 255.272,A -85,B 0,C 180,E1 -6583.211,E2 -6583.211} C_VEL
LIN {X 0,Y 490.188,Z 242.637,A -85,B 0,C 180,E1 -6583.788,E2 -6583.788} C_VEL
LIN {X 0,Y 490.18,Z 232.739,A -85,B 0,C 180,E1 -6584.119,E2 -6584.119} C_VEL
LIN {X 0,Y 488.679,Z 220.623,A -85,B 0,C 180,E1 -6584.442,E2 -6584.442} C_VEL
LIN {X 0,Y 489.22,Z 204.232,A -85,B 0,C 180,E1 -6587.989,E2 -6587.989} C_VEL
LIN {X 0,Y 489.762,Z 188.5,A -85,B 0,C 180,E1 -6591.462,E2 -6591.462} C_VEL
LIN {X 0,Y 490.461,Z 174.832,A -85,B 0,C 180,E1 -6594.552,E2 -6594.552} C_VEL
LIN {X 0,Y 490.957,Z 165.11,A -85,B 0,C 180,E1 -6596.801,E2 -6596.801} C_VEL
LIN {X 0,Y 490.634,Z 161.14,A -85,B 0,C 180,E1 -6597.76,E2 -6597.76} C_VEL
LIN {X 0,Y 488.716,Z 151.612,A -85,B 0,C 180,E1 -6600.218,E2 -6600.218} C_VEL
LIN {X 0,Y 488.73,Z 151.607,A -85,B 0,C 180,E1 -6603.483,E2 -6603.483} C_VEL
LIN {X 0,Y 488.683,Z 151.612,A -85,B 0,C 180,E1 -6606.354,E2 -6606.354} C_VEL
LIN {X 0,Y 488.691,Z 151.613,A -85,B 0,C 180,E1 -6609.253,E2 -6609.253} C_VEL
LIN {X 0,Y 488.687,Z 151.609,A -85,B 0,C 180,E1 -6611.597,E2 -6611.597} C_VEL
LIN {X 0,Y 488.703,Z 151.609,A -85,B 0,C 180,E1 -6614.8,E2 -6614.8} C_VEL
LIN {X 0,Y 488.726,Z 151.609,A -85,B 0,C 180,E1 -6617.478,E2 -6617.478} C_VEL
LIN {X 0,Y 488.738,Z 151.609,A -85,B 0,C 180,E1 -6620.749,E2 -6620.749} C_VEL
LIN {X 0,Y 488.657,Z 151.616,A -85,B 0,C 180,E1 -6623.866,E2 -6623.866} C_VEL
LIN {X 0,Y 488.727,Z 151.606,A -85,B 0,C 180,E1 -6626.876,E2 -6626.876} C_VEL
LIN {X 0,Y 488.722,Z 151.608,A -85,B 0,C 180,E1 -6629.78,E2 -6629.78} C_VEL
LIN {X 0,Y 488.786,Z 151.6,A -85,B 0,C 180,E1 -6633.054,E2 -6633.054} C_VEL
LIN {X 0,Y 488.67,Z 151.614,A -85,B 0,C 180,E1 -6636.253,E2 -6636.253} C_VEL
LIN {X 0,Y 488.732,Z 151.607,A -85,B 0,C 180,E1 -6639.175,E2 -6639.175} C_VEL
LIN {X 0,Y 488.722,Z 151.609,A -85,B 0,C 180,E1 -6642.423,E2 -6642.423} C_VEL
LIN {X 0,Y 488.748,Z 151.604,A -85,B 0,C 180,E1 -6644.999,E2 -6644.999} C_VEL
LIN {X 0,Y 488.815,Z 151.594,A -85,B 0,C 180,E1 -6648.388,E2 -6648.388} C_VEL
LIN {X 0,Y 488.799,Z 151.597,A -85,B 0,C 180,E1 -6651.733,E2 -6651.733} C_VEL
LIN {X 0,Y 488.847,Z 151.593,A -85,B 0,C 180,E1 -6654.224,E2 -6654.224} C_VEL
LIN {X 0,Y 488.949,Z 151.582,A -85,B 0,C 180,E1 -6657.529,E2 -6657.529} C_VEL
LIN {X 0,Y 488.951,Z 151.578,A -85,B 0,C 180,E1 -6660,E2 -6660} C_VEL
LIN {X 0,Y 488.939,Z 151.58,A -85,B 0,C 180,E1 -6662.471,E2 -6662.471} C_VEL
LIN {X 0,Y 488.84,Z 151.593,A -85,B 0,C 180,E1 -6665.776,E2 -6665.776} C_VEL
LIN {X 0,Y 488.804,Z 151.599,A -85,B 0,C 180,E1 -6668.267,E2 -6668.267} C_VEL
LIN {X 0,Y 488.816,Z 151.597,A -85,B 0,C 180,E1 -6671.612,E2 -6671.612} C_VEL
LIN {X 0,Y 488.749,Z 151.603,A -85,B 0,C 180,E1 -6675.001,E2 -6675.001} C_VEL
LIN {X 0,Y 488.74,Z 151.605,A -85,B 0,C 180,E1 -6678.443,E2 -6678.443} C_VEL
LIN {X 0,Y 488.727,Z 151.609,A -85,B 0,C 180,E1 -6681.07,E2 -6681.07} C_VEL
LIN {X 0,Y 488.686,Z 151.611,A -85,B 0,C 180,E1 -6683.746,E2 -6683.746} C_VEL
LIN {X 0,Y 488.705,Z 151.611,A -85,B 0,C 180,E1 -6686.475,E2 -6686.475} C_VEL
LIN {X 0,Y 488.697,Z 151.61,A -85,B 0,C 180,E1 -6689.272,E2 -6689.272} C_VEL
LIN {X 0,Y 488.693,Z 151.61,A -85,B 0,C 180,E1 -6692.148,E2 -6692.148} C_VEL
LIN {X 0,Y 488.712,Z 151.61,A -85,B 0,C 180,E1 -6695.116,E2 -6695.116} C_VEL
LIN {X 0,Y 488.668,Z 151.616,A -85,B 0,C 180,E1 -6698.201,E2 -6698.201} C_VEL
LIN {X 0,Y 488.707,Z 151.607,A -85,B 0,C 180,E1 -6700.346,E2 -6700.346} C_VEL
LIN {X 0,Y 488.677,Z 151.613,A -85,B 0,C 180,E1 -6703.656,E2 -6703.656} C_VEL
LIN {X 0,Y 488.683,Z 151.614,A -85,B 0,C 180,E1 -6706.348,E2 -6706.348} C_VEL
LIN {X 0,Y 488.71,Z 151.61,A -85,B 0,C 180,E1 -6708.587,E2 -6708.587} C_VEL
LIN {X 0,Y 488.67,Z 151.614,A -85,B 0,C 180,E1 -6711.801,E2 -6711.801} C_VEL
LIN {X 0,Y 488.715,Z 151.611,A -85,B 0,C 180,E1 -6715.054,E2 -6715.054} C_VEL
LIN {X 0,Y 488.701,Z 151.612,A -85,B 0,C 180,E1 -6718.047,E2 -6718.047} C_VEL
LIN {X 0,Y 488.727,Z 151.606,A -85,B 0,C 180,E1 -6720.776,E2 -6720.776} C_VEL
LIN {X 0,Y 488.73,Z 151.607,A -85,B 0,C 180,E1 -6723.528,E2 -6723.528} C_VEL
LIN {X 0,Y 488.701,Z 151.609,A -85,B 0,C 180,E1 -6724.366,E2 -6724.366} C_VEL
LIN {X 0,Y 488.053,Z 151.693,A -85,B 0,C 180,E1 -6725.054,E2 -6725.054} C_VEL
LIN {X 0,Y 485.196,Z 152.048,A -85,B 0,C 180,E1 -6726.171,E2 -6726.171} C_VEL
LIN {X 0,Y 482.766,Z 152.349,A -85,B 0,C 180,E1 -6727.071,E2 -6727.071} C_VEL
LIN {X 0,Y 481.717,Z 152.479,A -85,B 0,C 180,E1 -6727.767,E2 -6727.767} C_VEL
LIN {X 0,Y 481.63,Z 152.489,A -85,B 0,C 180,E1 -6728.003,E2 -6728.003} C_VEL
LIN {X 0,Y 481.703,Z 152.483,A -85,B 0,C 180,E1 -6730.395,E2 -6730.395} C_VEL
LIN {X 0,Y 481.689,Z 152.486,A -85,B 0,C 180,E1 -6733.035,E2 -6733.035} C_VEL
LIN {X 0,Y 481.68,Z 152.484,A -85,B 0,C 180,E1 -6735.64,E2 -6735.64} C_VEL
LIN {X 0,Y 481.75,Z 152.478,A -85,B 0,C 180,E1 -6738.217,E2 -6738.217} C_VEL
LIN {X 0,Y 481.761,Z 152.476,A -85,B 0,C 180,E1 -6741.613,E2 -6741.613} C_VEL
LIN {X 0,Y 481.817,Z 152.467,A -85,B 0,C 180,E1 -6744.141,E2 -6744.141} C_VEL
LIN {X 0,Y 481.929,Z 152.453,A -85,B 0,C 180,E1 -6747.494,E2 -6747.494} C_VEL
LIN {X 0,Y 481.912,Z 152.459,A -85,B 0,C 180,E1 -6750.001,E2 -6750.001} C_VEL
LIN {X 0,Y 481.921,Z 152.453,A -85,B 0,C 180,E1 -6752.509,E2 -6752.509} C_VEL
LIN {X 0,Y 481.818,Z 152.467,A -85,B 0,C 180,E1 -6755.862,E2 -6755.862} C_VEL
LIN {X 0,Y 481.765,Z 152.476,A -85,B 0,C 180,E1 -6758.389,E2 -6758.389} C_VEL
LIN {X 0,Y 481.755,Z 152.479,A -85,B 0,C 180,E1 -6761.786,E2 -6761.786} C_VEL
LIN {X 0,Y 481.741,Z 152.48,A -85,B 0,C 180,E1 -6765.225,E2 -6765.225} C_VEL
LIN {X 0,Y 481.713,Z 152.483,A -85,B 0,C 180,E1 -6768.723,E2 -6768.723} C_VEL
LIN {X 0,Y 481.65,Z 152.489,A -85,B 0,C 180,E1 -6771.396,E2 -6771.396} C_VEL
LIN {X 0,Y 481.652,Z 152.488,A -85,B 0,C 180,E1 -6774.116,E2 -6774.116} C_VEL
LIN {X 0,Y 481.657,Z 152.49,A -85,B 0,C 180,E1 -6777.118,E2 -6777.118} C_VEL
LIN {X 0,Y 481.671,Z 152.485,A -85,B 0,C 180,E1 -6779.743,E2 -6779.743} C_VEL
LIN {X 0,Y 481.675,Z 152.485,A -85,B 0,C 180,E1 -6782.675,E2 -6782.675} C_VEL
LIN {X 0,Y 481.633,Z 152.491,A -85,B 0,C 180,E1 -6785.711,E2 -6785.711} C_VEL
LIN {X 0,Y 481.632,Z 152.493,A -85,B 0,C 180,E1 -6788.864,E2 -6788.864} C_VEL
LIN {X 0,Y 481.64,Z 152.491,A -85,B 0,C 180,E1 -6791.911,E2 -6791.911} C_VEL
LIN {X 0,Y 481.659,Z 152.487,A -85,B 0,C 180,E1 -6794.459,E2 -6794.459} C_VEL
LIN {X 0,Y 481.653,Z 152.487,A -85,B 0,C 180,E1 -6797.84,E2 -6797.84} C_VEL
LIN {X 0,Y 481.656,Z 152.489,A -85,B 0,C 180,E1 -6800.656,E2 -6800.656} C_VEL
LIN {X 0,Y 481.622,Z 152.491,A -85,B 0,C 180,E1 -6803.378,E2 -6803.378} C_VEL
LIN {X 0,Y 481.681,Z 152.484,A -85,B 0,C 180,E1 -6806.328,E2 -6806.328} C_VEL
LIN {X 0,Y 481.766,Z 152.536,A -85,B 0,C 180,E1 -6808.23,E2 -6808.23} C_VEL
LIN {X 0,Y 482.352,Z 157.81,A -85,B 0,C 180,E1 -6810.305,E2 -6810.305} C_VEL
LIN {X 0,Y 482.054,Z 166.511,A -85,B 0,C 180,E1 -6813.598,E2 -6813.598} C_VEL
LIN {X 0,Y 481.824,Z 173.916,A -85,B 0,C 180,E1 -6816.352,E2 -6816.352} C_VEL
LIN {X 0,Y 481.62,Z 182.48,A -85,B 0,C 180,E1 -6819.499,E2 -6819.499} C_VEL
LIN {X 0,Y 481.416,Z 192.251,A -85,B 0,C 180,E1 -6823.024,E2 -6823.024} C_VEL
LIN {X 0,Y 481.235,Z 200.741,A -85,B 0,C 180,E1 -6826.056,E2 -6826.056} C_VEL
LIN {X 0,Y 481.099,Z 209.25,A -85,B 0,C 180,E1 -6829.053,E2 -6829.053} C_VEL
LIN {X 0,Y 481.052,Z 214.959,A -85,B 0,C 180,E1 -6831.044,E2 -6831.044} C_VEL
LIN {X 0,Y 482.172,Z 225.606,A -85,B 0,C 180,E1 -6831.513,E2 -6831.513} C_VEL
LIN {X 0,Y 481.936,Z 235.982,A -85,B 0,C 180,E1 -6832.142,E2 -6832.142} C_VEL
LIN {X 0,Y 481.689,Z 244.238,A -85,B 0,C 180,E1 -6832.817,E2 -6832.817} C_VEL
LIN {X 0,Y 481.414,Z 252.644,A -85,B 0,C 180,E1 -6833.714,E2 -6833.714} C_VEL
LIN {X 0,Y 481.369,Z 258.729,A -85,B 0,C 180,E1 -6834.554,E2 -6834.554} C_VEL
LIN {X 0,Y 481.176,Z 264.609,A -85,B 0,C 180,E1 -6835.602,E2 -6835.602} C_VEL
LIN {X 0,Y 481.099,Z 268.949,A -85,B 0,C 180,E1 -6836.65,E2 -6836.65} C_VEL
LIN {X 0,Y 480.966,Z 271.509,A -85,B 0,C 180,E1 -6837.488,E2 -6837.488} C_VEL
LIN {X 0,Y 480.842,Z 273.323,A -85,B 0,C 180,E1 -6838.325,E2 -6838.325} C_VEL
LIN {X 0,Y 480.788,Z 274.433,A -85,B 0,C 180,E1 -6839.163,E2 -6839.163} C_VEL
LIN {X 0,Y 480.776,Z 274.868,A -85,B 0,C 180,E1 -6840,E2 -6840} C_VEL
LIN {X 0,Y 480.789,Z 274.632,A -85,B 0,C 180,E1 -6840.838,E2 -6840.838} C_VEL
LIN {X 0,Y 480.844,Z 273.725,A -85,B 0,C 180,E1 -6841.675,E2 -6841.675} C_VEL
LIN {X 0,Y 481.027,Z 271.059,A -85,B 0,C 180,E1 -6842.931,E2 -6842.931} C_VEL
LIN {X 0,Y 481.197,Z 268.337,A -85,B 0,C 180,E1 -6843.768,E2 -6843.768} C_VEL
LIN {X 0,Y 481.299,Z 263.764,A -85,B 0,C 180,E1 -6844.816,E2 -6844.816} C_VEL
LIN {X 0,Y 481.354,Z 257.612,A -85,B 0,C 180,E1 -6845.866,E2 -6845.866} C_VEL
LIN {X 0,Y 481.618,Z 250.06,A -85,B 0,C 180,E1 -6846.837,E2 -6846.837} C_VEL
LIN {X 0,Y 481.902,Z 241.838,A -85,B 0,C 180,E1 -6847.648,E2 -6847.648} C_VEL
LIN {X 0,Y 482.234,Z 233.634,A -85,B 0,C 180,E1 -6848.275,E2 -6848.275} C_VEL
LIN {X 0,Y 482.283,Z 224.701,A -85,B 0,C 180,E1 -6848.801,E2 -6848.801} C_VEL
LIN {X 0,Y 481.099,Z 215.431,A -85,B 0,C 180,E1 -6849.247,E2 -6849.247} C_VEL
LIN {X 0,Y 481.235,Z 207.087,A -85,B 0,C 180,E1 -6852.225,E2 -6852.225} C_VEL
LIN {X 0,Y 481.492,Z 197.84,A -85,B 0,C 180,E1 -6855.557,E2 -6855.557} C_VEL
LIN {X 0,Y 481.703,Z 189.236,A -85,B 0,C 180,E1 -6858.722,E2 -6858.722} C_VEL
LIN {X 0,Y 481.921,Z 180.966,A -85,B 0,C 180,E1 -6861.831,E2 -6861.831} C_VEL
LIN {X 0,Y 482.202,Z 172.769,A -85,B 0,C 180,E1 -6865.003,E2 -6865.003} C_VEL
LIN {X 0,Y 482.644,Z 165.83,A -85,B 0,C 180,E1 -6867.773,E2 -6867.773} C_VEL
LIN {X 0,Y 482.914,Z 160.114,A -85,B 0,C 180,E1 -6870.138,E2 -6870.138} C_VEL
LIN {X 0,Y 482.168,Z 154.685,A -85,B 0,C 180,E1 -6872.637,E2 -6872.637} C_VEL
LIN {X 0,Y 481.681,Z 152.488,A -85,B 0,C 180,E1 -6873.785,E2 -6873.785} C_VEL
LIN {X 0,Y 481.631,Z 152.495,A -85,B 0,C 180,E1 -6876.747,E2 -6876.747} C_VEL
LIN {X 0,Y 481.683,Z 152.487,A -85,B 0,C 180,E1 -6879.94,E2 -6879.94} C_VEL
LIN {X 0,Y 481.638,Z 152.493,A -85,B 0,C 180,E1 -6883.147,E2 -6883.147} C_VEL
LIN {X 0,Y 481.66,Z 152.49,A -85,B 0,C 180,E1 -6885.641,E2 -6885.641} C_VEL
LIN {X 0,Y 481.662,Z 152.49,A -85,B 0,C 180,E1 -6888.958,E2 -6888.958} C_VEL
LIN {X 0,Y 481.66,Z 152.49,A -85,B 0,C 180,E1 -6891.992,E2 -6891.992} C_VEL
LIN {X 0,Y 481.691,Z 152.487,A -85,B 0,C 180,E1 -6895.317,E2 -6895.317} C_VEL
LIN {X 0,Y 481.678,Z 152.543,A -85,B 0,C 180,E1 -6897.466,E2 -6897.466} C_VEL
LIN {X 0,Y 483.087,Z 158.904,A -85,B 0,C 180,E1 -6899.872,E2 -6899.872} C_VEL
LIN {X 0,Y 484.534,Z 166.124,A -85,B 0,C 180,E1 -6902.225,E2 -6902.225} C_VEL
LIN {X 0,Y 484.534,Z 169.733,A -85,B 0,C 180,E1 -6903.278,E2 -6903.278} C_VEL
LIN {X 0,Y 483.483,Z 181.384,A -85,B 0,C 180,E1 -6906.317,E2 -6906.317} C_VEL
LIN {X 0,Y 482.632,Z 194.635,A -85,B 0,C 180,E1 -6909.543,E2 -6909.543} C_VEL
LIN {X 0,Y 482.115,Z 206.015,A -85,B 0,C 180,E1 -6912.173,E2 -6912.173} C_VEL
LIN {X 0,Y 481.628,Z 220.657,A -85,B 0,C 180,E1 -6915.433,E2 -6915.433} C_VEL
LIN {X 0,Y 483.267,Z 234.787,A -85,B 0,C 180,E1 -6915.82,E2 -6915.82} C_VEL
LIN {X 0,Y 483.092,Z 246.827,A -85,B 0,C 180,E1 -6916.271,E2 -6916.271} C_VEL
LIN {X 0,Y 482.702,Z 258.155,A -85,B 0,C 180,E1 -6916.849,E2 -6916.849} C_VEL
LIN {X 0,Y 482.32,Z 270.209,A -85,B 0,C 180,E1 -6917.652,E2 -6917.652} C_VEL
LIN {X 0,Y 482.012,Z 280.754,A -85,B 0,C 180,E1 -6918.54,E2 -6918.54} C_VEL
LIN {X 0,Y 481.664,Z 289.896,A -85,B 0,C 180,E1 -6919.49,E2 -6919.49} C_VEL
LIN {X 0,Y 481.398,Z 298.258,A -85,B 0,C 180,E1 -6920.546,E2 -6920.546} C_VEL
LIN {X 0,Y 481.162,Z 306.425,A -85,B 0,C 180,E1 -6921.811,E2 -6921.811} C_VEL
LIN {X 0,Y 481.011,Z 311.937,A -85,B 0,C 180,E1 -6922.865,E2 -6922.865} C_VEL
LIN {X 0,Y 480.93,Z 317.316,A -85,B 0,C 180,E1 -6924.127,E2 -6924.127} C_VEL
LIN {X 0,Y 480.848,Z 321.477,A -85,B 0,C 180,E1 -6925.388,E2 -6925.388} C_VEL
LIN {X 0,Y 480.896,Z 324.548,A -85,B 0,C 180,E1 -6926.647,E2 -6926.647} C_VEL
LIN {X 0,Y 480.87,Z 326.024,A -85,B 0,C 180,E1 -6927.486,E2 -6927.486} C_VEL
LIN {X 0,Y 480.825,Z 327.065,A -85,B 0,C 180,E1 -6928.324,E2 -6928.324} C_VEL
LIN {X 0,Y 480.768,Z 327.706,A -85,B 0,C 180,E1 -6929.161,E2 -6929.161} C_VEL
LIN {X 0,Y 480.758,Z 327.944,A -85,B 0,C 180,E1 -6929.999,E2 -6929.999} C_VEL
LIN {X 0,Y 480.767,Z 327.733,A -85,B 0,C 180,E1 -6930.836,E2 -6930.836} C_VEL
LIN {X 0,Y 480.824,Z 327.124,A -85,B 0,C 180,E1 -6931.674,E2 -6931.674} C_VEL
LIN {X 0,Y 480.869,Z 326.117,A -85,B 0,C 180,E1 -6932.512,E2 -6932.512} C_VEL
LIN {X 0,Y 480.894,Z 324.666,A -85,B 0,C 180,E1 -6933.35,E2 -6933.35} C_VEL
LIN {X 0,Y 480.84,Z 321.642,A -85,B 0,C 180,E1 -6934.61,E2 -6934.61} C_VEL
LIN {X 0,Y 480.929,Z 317.534,A -85,B 0,C 180,E1 -6935.87,E2 -6935.87} C_VEL
LIN {X 0,Y 481.096,Z 311.205,A -85,B 0,C 180,E1 -6937.342,E2 -6937.342} C_VEL
LIN {X 0,Y 481.248,Z 304.274,A -85,B 0,C 180,E1 -6938.607,E2 -6938.607} C_VEL
LIN {X 0,Y 481.472,Z 295.537,A -85,B 0,C 180,E1 -6939.874,E2 -6939.874} C_VEL
LIN {X 0,Y 481.84,Z 285.575,A -85,B 0,C 180,E1 -6941.035,E2 -6941.035} C_VEL
LIN {X 0,Y 482.199,Z 275.848,A -85,B 0,C 180,E1 -6941.948,E2 -6941.948} C_VEL
LIN {X 0,Y 482.557,Z 264.04,A -85,B 0,C 180,E1 -6942.831,E2 -6942.831} C_VEL
LIN {X 0,Y 482.958,Z 252.251,A -85,B 0,C 180,E1 -6943.516,E2 -6943.516} C_VEL
LIN {X 0,Y 483.263,Z 239.21,A -85,B 0,C 180,E1 -6944.07,E2 -6944.07} C_VEL
LIN {X 0,Y 483.116,Z 232.56,A -85,B 0,C 180,E1 -6944.29,E2 -6944.29} C_VEL
LIN {X 0,Y 481.65,Z 220.617,A -85,B 0,C 180,E1 -6944.604,E2 -6944.604} C_VEL
LIN {X 0,Y 482.116,Z 205.98,A -85,B 0,C 180,E1 -6947.824,E2 -6947.824} C_VEL
LIN {X 0,Y 482.745,Z 190.3,A -85,B 0,C 180,E1 -6951.342,E2 -6951.342} C_VEL
LIN {X 0,Y 483.47,Z 176.681,A -85,B 0,C 180,E1 -6954.473,E2 -6954.473} C_VEL
LIN {X 0,Y 484.026,Z 165.178,A -85,B 0,C 180,E1 -6957.179,E2 -6957.179} C_VEL
LIN {X 0,Y 483.018,Z 159.19,A -85,B 0,C 180,E1 -6958.694,E2 -6958.694} C_VEL
LIN {X 0,Y 481.67,Z 152.489,A -85,B 0,C 180,E1 -6960.452,E2 -6960.452} C_VEL
LIN {X 0,Y 481.691,Z 152.486,A -85,B 0,C 180,E1 -6963.732,E2 -6963.732} C_VEL
LIN {X 0,Y 481.623,Z 152.492,A -85,B 0,C 180,E1 -6966.745,E2 -6966.745} C_VEL
LIN {X 0,Y 481.65,Z 152.487,A -85,B 0,C 180,E1 -6969.941,E2 -6969.941} C_VEL
LIN {X 0,Y 481.619,Z 152.491,A -85,B 0,C 180,E1 -6973.145,E2 -6973.145} C_VEL
LIN {X 0,Y 481.65,Z 152.489,A -85,B 0,C 180,E1 -6975.639,E2 -6975.639} C_VEL
LIN {X 0,Y 481.664,Z 152.487,A -85,B 0,C 180,E1 -6978.083,E2 -6978.083} C_VEL
LIN {X 0,Y 481.692,Z 152.484,A -85,B 0,C 180,E1 -6981.143,E2 -6981.143} C_VEL
LIN {X 0,Y 481.648,Z 152.487,A -85,B 0,C 180,E1 -6984.795,E2 -6984.795} C_VEL
LIN {X 0,Y 481.661,Z 152.488,A -85,B 0,C 180,E1 -6987.325,E2 -6987.325} C_VEL
LIN {X 0,Y 481.676,Z 152.485,A -85,B 0,C 180,E1 -6990.259,E2 -6990.259} C_VEL
LIN {X 0,Y 481.739,Z 152.478,A -85,B 0,C 180,E1 -6993.112,E2 -6993.112} C_VEL
LIN {X 0,Y 481.656,Z 152.491,A -85,B 0,C 180,E1 -6995.886,E2 -6995.886} C_VEL
LIN {X 0,Y 481.688,Z 152.484,A -85,B 0,C 180,E1 -6999.027,E2 -6999.027} C_VEL
LIN {X 0,Y 481.694,Z 152.483,A -85,B 0,C 180,E1 -7002.158,E2 -7002.158} C_VEL
LIN {X 0,Y 481.728,Z 152.48,A -85,B 0,C 180,E1 -7004.775,E2 -7004.775} C_VEL
LIN {X 0,Y 481.779,Z 152.471,A -85,B 0,C 180,E1 -7008.216,E2 -7008.216} C_VEL
LIN {X 0,Y 481.745,Z 152.476,A -85,B 0,C 180,E1 -7011.611,E2 -7011.611} C_VEL
LIN {X 0,Y 481.807,Z 152.47,A -85,B 0,C 180,E1 -7014.139,E2 -7014.139} C_VEL
LIN {X 0,Y 481.916,Z 152.457,A -85,B 0,C 180,E1 -7017.492,E2 -7017.492} C_VEL
LIN {X 0,Y 481.922,Z 152.454,A -85,B 0,C 180,E1 -7020,E2 -7020} C_VEL
LIN {X 0,Y 481.907,Z 152.456,A -85,B 0,C 180,E1 -7022.508,E2 -7022.508} C_VEL
LIN {X 0,Y 481.801,Z 152.47,A -85,B 0,C 180,E1 -7025.861,E2 -7025.861} C_VEL
LIN {X 0,Y 481.75,Z 152.477,A -85,B 0,C 180,E1 -7028.388,E2 -7028.388} C_VEL
LIN {X 0,Y 481.781,Z 152.472,A -85,B 0,C 180,E1 -7031.784,E2 -7031.784} C_VEL
LIN {X 0,Y 481.729,Z 152.476,A -85,B 0,C 180,E1 -7035.225,E2 -7035.225} C_VEL
LIN {X 0,Y 481.698,Z 152.482,A -85,B 0,C 180,E1 -7038.722,E2 -7038.722} C_VEL
LIN {X 0,Y 481.658,Z 152.489,A -85,B 0,C 180,E1 -7041.394,E2 -7041.394} C_VEL
LIN {X 0,Y 481.665,Z 152.487,A -85,B 0,C 180,E1 -7044.114,E2 -7044.114} C_VEL
LIN {X 0,Y 481.68,Z 152.482,A -85,B 0,C 180,E1 -7047.128,E2 -7047.128} C_VEL
LIN {X 0,Y 481.661,Z 152.49,A -85,B 0,C 180,E1 -7049.742,E2 -7049.742} C_VEL
LIN {X 0,Y 481.661,Z 152.488,A -85,B 0,C 180,E1 -7052.675,E2 -7052.675} C_VEL
LIN {X 0,Y 481.631,Z 152.49,A -85,B 0,C 180,E1 -7055.71,E2 -7055.71} C_VEL
LIN {X 0,Y 481.658,Z 152.485,A -85,B 0,C 180,E1 -7058.86,E2 -7058.86} C_VEL
LIN {X 0,Y 481.642,Z 152.489,A -85,B 0,C 180,E1 -7061.914,E2 -7061.914} C_VEL
LIN {X 0,Y 481.65,Z 152.49,A -85,B 0,C 180,E1 -7064.459,E2 -7064.459} C_VEL
LIN {X 0,Y 481.645,Z 152.491,A -85,B 0,C 180,E1 -7067.841,E2 -7067.841} C_VEL
LIN {X 0,Y 481.652,Z 152.487,A -85,B 0,C 180,E1 -7070.655,E2 -7070.655} C_VEL
LIN {X 0,Y 481.617,Z 152.494,A -85,B 0,C 180,E1 -7073.378,E2 -7073.378} C_VEL
LIN {X 0,Y 481.703,Z 152.483,A -85,B 0,C 180,E1 -7076.332,E2 -7076.332} C_VEL
LIN {X 0,Y 481.653,Z 152.489,A -85,B 0,C 180,E1 -7079.417,E2 -7079.417} C_VEL
LIN {X 0,Y 481.69,Z 152.483,A -85,B 0,C 180,E1 -7082.169,E2 -7082.169} C_VEL
LIN {X 0,Y 481.671,Z 152.489,A -85,B 0,C 180,E1 -7084.969,E2 -7084.969} C_VEL
LIN {X 0,Y 481.63,Z 152.489,A -85,B 0,C 180,E1 -7088.003,E2 -7088.003} C_VEL
LIN {X 0,Y 480.965,Z 152.575,A -85,B 0,C 180,E1 -7088.701,E2 -7088.701} C_VEL
LIN {X 0,Y 478.138,Z 152.927,A -85,B 0,C 180,E1 -7089.835,E2 -7089.835} C_VEL
LIN {X 0,Y 475.754,Z 153.224,A -85,B 0,C 180,E1 -7090.749,E2 -7090.749} C_VEL
LIN {X 0,Y 474.734,Z 153.351,A -85,B 0,C 180,E1 -7091.455,E2 -7091.455} C_VEL
LIN {X 0,Y 474.653,Z 153.361,A -85,B 0,C 180,E1 -7091.694,E2 -7091.694} C_VEL
LIN {X 0,Y 474.698,Z 153.355,A -85,B 0,C 180,E1 -7094.546,E2 -7094.546} C_VEL
LIN {X 0,Y 474.703,Z 153.354,A -85,B 0,C 180,E1 -7098.039,E2 -7098.039} C_VEL
LIN {X 0,Y 474.726,Z 153.351,A -85,B 0,C 180,E1 -7101.488,E2 -7101.488} C_VEL
LIN {X 0,Y 474.78,Z 153.344,A -85,B 0,C 180,E1 -7104.054,E2 -7104.054} C_VEL
LIN {X 0,Y 474.895,Z 153.329,A -85,B 0,C 180,E1 -7107.457,E2 -7107.457} C_VEL
LIN {X 0,Y 474.882,Z 153.335,A -85,B 0,C 180,E1 -7110.001,E2 -7110.001} C_VEL
LIN {X 0,Y 474.887,Z 153.329,A -85,B 0,C 180,E1 -7112.546,E2 -7112.546} C_VEL
LIN {X 0,Y 474.781,Z 153.344,A -85,B 0,C 180,E1 -7115.949,E2 -7115.949} C_VEL
LIN {X 0,Y 474.73,Z 153.352,A -85,B 0,C 180,E1 -7118.515,E2 -7118.515} C_VEL
LIN {X 0,Y 474.708,Z 153.355,A -85,B 0,C 180,E1 -7121.964,E2 -7121.964} C_VEL
LIN {X 0,Y 474.684,Z 153.356,A -85,B 0,C 180,E1 -7125.768,E2 -7125.768} C_VEL
LIN {X 0,Y 474.667,Z 153.359,A -85,B 0,C 180,E1 -7129.011,E2 -7129.011} C_VEL
LIN {X 0,Y 474.593,Z 153.371,A -85,B 0,C 180,E1 -7131.73,E2 -7131.73} C_VEL
LIN {X 0,Y 474.63,Z 153.361,A -85,B 0,C 180,E1 -7134.496,E2 -7134.496} C_VEL
LIN {X 0,Y 474.604,Z 153.367,A -85,B 0,C 180,E1 -7137.327,E2 -7137.327} C_VEL
LIN {X 0,Y 474.602,Z 153.368,A -85,B 0,C 180,E1 -7140.232,E2 -7140.232} C_VEL
LIN {X 0,Y 474.63,Z 153.364,A -85,B 0,C 180,E1 -7143.222,E2 -7143.222} C_VEL
LIN {X 0,Y 474.585,Z 153.367,A -85,B 0,C 180,E1 -7146.325,E2 -7146.325} C_VEL
LIN {X 0,Y 474.603,Z 153.364,A -85,B 0,C 180,E1 -7149.644,E2 -7149.644} C_VEL
LIN {X 0,Y 474.594,Z 153.371,A -85,B 0,C 180,E1 -7152.233,E2 -7152.233} C_VEL
LIN {X 0,Y 474.622,Z 153.366,A -85,B 0,C 180,E1 -7155.298,E2 -7155.298} C_VEL
LIN {X 0,Y 474.626,Z 153.363,A -85,B 0,C 180,E1 -7158.215,E2 -7158.215} C_VEL
LIN {X 0,Y 474.631,Z 153.366,A -85,B 0,C 180,E1 -7160.453,E2 -7160.453} C_VEL
LIN {X 0,Y 474.585,Z 153.369,A -85,B 0,C 180,E1 -7163.676,E2 -7163.676} C_VEL
LIN {X 0,Y 474.637,Z 153.363,A -85,B 0,C 180,E1 -7166.779,E2 -7166.779} C_VEL
LIN {X 0,Y 474.679,Z 153.415,A -85,B 0,C 180,E1 -7168.104,E2 -7168.104} C_VEL
LIN {X 0,Y 475.326,Z 157.675,A -85,B 0,C 180,E1 -7169.82,E2 -7169.82} C_VEL
LIN {X 0,Y 475.119,Z 165.193,A -85,B 0,C 180,E1 -7172.706,E2 -7172.706} C_VEL
LIN {X 0,Y 474.823,Z 173.863,A -85,B 0,C 180,E1 -7175.981,E2 -7175.981} C_VEL
LIN {X 0,Y 474.605,Z 182.478,A -85,B 0,C 180,E1 -7179.182,E2 -7179.182} C_VEL
LIN {X 0,Y 474.382,Z 191.034,A -85,B 0,C 180,E1 -7182.32,E2 -7182.32} C_VEL
LIN {X 0,Y 474.206,Z 199.58,A -85,B 0,C 180,E1 -7185.407,E2 -7185.407} C_VEL
LIN {X 0,Y 474.083,Z 208.175,A -85,B 0,C 180,E1 -7188.478,E2 -7188.478} C_VEL
LIN {X 0,Y 473.966,Z 214.957,A -85,B 0,C 180,E1 -7190.882,E2 -7190.882} C_VEL
LIN {X 0,Y 475.154,Z 225.962,A -85,B 0,C 180,E1 -7191.387,E2 -7191.387} C_VEL
LIN {X 0,Y 474.907,Z 236.263,A -85,B 0,C 180,E1 -7192.025,E2 -7192.025} C_VEL
LIN {X 0,Y 474.626,Z 245.406,A -85,B 0,C 180,E1 -7192.798,E2 -7192.798} C_VEL
LIN {X 0,Y 474.384,Z 252.908,A -85,B 0,C 180,E1 -7193.621,E2 -7193.621} C_VEL
LIN {X 0,Y 474.314,Z 259.008,A -85,B 0,C 180,E1 -7194.473,E2 -7194.473} C_VEL
LIN {X 0,Y 474.129,Z 264.909,A -85,B 0,C 180,E1 -7195.537,E2 -7195.537} C_VEL
LIN {X 0,Y 474.027,Z 269.273,A -85,B 0,C 180,E1 -7196.6,E2 -7196.6} C_VEL
LIN {X 0,Y 473.893,Z 271.852,A -85,B 0,C 180,E1 -7197.45,E2 -7197.45} C_VEL
LIN {X 0,Y 473.777,Z 273.684,A -85,B 0,C 180,E1 -7198.3,E2 -7198.3} C_VEL
LIN {X 0,Y 473.715,Z 274.814,A -85,B 0,C 180,E1 -7199.15,E2 -7199.15} C_VEL
LIN {X 0,Y 473.701,Z 275.267,A -85,B 0,C 180,E1 -7200,E2 -7200} C_VEL
LIN {X 0,Y 473.717,Z 275.049,A -85,B 0,C 180,E1 -7200.85,E2 -7200.85} C_VEL
LIN {X 0,Y 473.779,Z 274.159,A -85,B 0,C 180,E1 -7201.7,E2 -7201.7} C_VEL
LIN {X 0,Y 473.974,Z 271.519,A -85,B 0,C 180,E1 -7202.975,E2 -7202.975} C_VEL
LIN {X 0,Y 474.146,Z 268.819,A -85,B 0,C 180,E1 -7203.825,E2 -7203.825} C_VEL
LIN {X 0,Y 474.261,Z 264.28,A -85,B 0,C 180,E1 -7204.888,E2 -7204.888} C_VEL
LIN {X 0,Y 474.324,Z 258.19,A -85,B 0,C 180,E1 -7205.953,E2 -7205.953} C_VEL
LIN {X 0,Y 474.589,Z 251.195,A -85,B 0,C 180,E1 -7206.885,E2 -7206.885} C_VEL
LIN {X 0,Y 474.927,Z 242.654,A -85,B 0,C 180,E1 -7207.761,E2 -7207.761} C_VEL
LIN {X 0,Y 475.274,Z 234.609,A -85,B 0,C 180,E1 -7208.397,E2 -7208.397} C_VEL
LIN {X 0,Y 475.385,Z 225.955,A -85,B 0,C 180,E1 -7208.93,E2 -7208.93} C_VEL
LIN {X 0,Y 474.243,Z 216.925,A -85,B 0,C 180,E1 -7209.382,E2 -7209.382} C_VEL
LIN {X 0,Y 474.04,Z 215.593,A -85,B 0,C 180,E1 -7209.44,E2 -7209.44} C_VEL
LIN {X 0,Y 474.194,Z 207.381,A -85,B 0,C 180,E1 -7212.41,E2 -7212.41} C_VEL
LIN {X 0,Y 474.45,Z 198.502,A -85,B 0,C 180,E1 -7215.666,E2 -7215.666} C_VEL
LIN {X 0,Y 474.699,Z 189.577,A -85,B 0,C 180,E1 -7219.009,E2 -7219.009} C_VEL
LIN {X 0,Y 474.943,Z 181.34,A -85,B 0,C 180,E1 -7222.169,E2 -7222.169} C_VEL
LIN {X 0,Y 475.229,Z 174.352,A -85,B 0,C 180,E1 -7224.928,E2 -7224.928} C_VEL
LIN {X 0,Y 475.663,Z 167.841,A -85,B 0,C 180,E1 -7227.561,E2 -7227.561} C_VEL
LIN {X 0,Y 476.002,Z 161.822,A -85,B 0,C 180,E1 -7230.132,E2 -7230.132} C_VEL
LIN {X 0,Y 475.47,Z 157.497,A -85,B 0,C 180,E1 -7232.149,E2 -7232.149} C_VEL
LIN {X 0,Y 474.674,Z 153.361,A -85,B 0,C 180,E1 -7234.366,E2 -7234.366} C_VEL
LIN {X 0,Y 474.596,Z 153.37,A -85,B 0,C 180,E1 -7237.383,E2 -7237.383} C_VEL
LIN {X 0,Y 474.633,Z 153.366,A -85,B 0,C 180,E1 -7239.647,E2 -7239.647} C_VEL
LIN {X 0,Y 474.612,Z 153.368,A -85,B 0,C 180,E1 -7242.935,E2 -7242.935} C_VEL
LIN {X 0,Y 474.612,Z 153.368,A -85,B 0,C 180,E1 -7245.894,E2 -7245.894} C_VEL
LIN {X 0,Y 474.634,Z 153.366,A -85,B 0,C 180,E1 -7249.04,E2 -7249.04} C_VEL
LIN {X 0,Y 474.616,Z 153.368,A -85,B 0,C 180,E1 -7251.704,E2 -7251.704} C_VEL
LIN {X 0,Y 474.629,Z 153.367,A -85,B 0,C 180,E1 -7254.725,E2 -7254.725} C_VEL
LIN {X 0,Y 474.628,Z 153.455,A -85,B 0,C 180,E1 -7256.831,E2 -7256.831} C_VEL
LIN {X 0,Y 476.107,Z 159.884,A -85,B 0,C 180,E1 -7259.423,E2 -7259.423} C_VEL
LIN {X 0,Y 477.599,Z 167.38,A -85,B 0,C 180,E1 -7261.997,E2 -7261.997} C_VEL
LIN {X 0,Y 477.616,Z 171.953,A -85,B 0,C 180,E1 -7263.332,E2 -7263.332} C_VEL
LIN {X 0,Y 476.458,Z 183.908,A -85,B 0,C 180,E1 -7266.529,E2 -7266.529} C_VEL
LIN {X 0,Y 475.626,Z 196.641,A -85,B 0,C 180,E1 -7269.68,E2 -7269.68} C_VEL
LIN {X 0,Y 475.042,Z 207.915,A -85,B 0,C 180,E1 -7272.344,E2 -7272.344} C_VEL
LIN {X 0,Y 474.616,Z 220.594,A -85,B 0,C 180,E1 -7275.227,E2 -7275.227} C_VEL
LIN {X 0,Y 476.265,Z 234.816,A -85,B 0,C 180,E1 -7275.634,E2 -7275.634} C_VEL
LIN {X 0,Y 476.128,Z 247.298,A -85,B 0,C 180,E1 -7276.12,E2 -7276.12} C_VEL
LIN {X 0,Y 475.68,Z 259.312,A -85,B 0,C 180,E1 -7276.76,E2 -7276.76} C_VEL
LIN {X 0,Y 475.289,Z 270.926,A -85,B 0,C 180,E1 -7277.562,E2 -7277.562} C_VEL
LIN {X 0,Y 474.962,Z 281.341,A -85,B 0,C 180,E1 -7278.476,E2 -7278.476} C_VEL
LIN {X 0,Y 474.562,Z 291.222,A -85,B 0,C 180,E1 -7279.547,E2 -7279.547} C_VEL
LIN {X 0,Y 474.304,Z 299.303,A -85,B 0,C 180,E1 -7280.618,E2 -7280.618} C_VEL
LIN {X 0,Y 474.075,Z 307.167,A -85,B 0,C 180,E1 -7281.903,E2 -7281.903} C_VEL
LIN {X 0,Y 473.901,Z 313.443,A -85,B 0,C 180,E1 -7283.185,E2 -7283.185} C_VEL
LIN {X 0,Y 473.861,Z 318.406,A -85,B 0,C 180,E1 -7284.467,E2 -7284.467} C_VEL
LIN {X 0,Y 473.76,Z 322.194,A -85,B 0,C 180,E1 -7285.745,E2 -7285.745} C_VEL
LIN {X 0,Y 473.822,Z 324.151,A -85,B 0,C 180,E1 -7286.597,E2 -7286.597} C_VEL
LIN {X 0,Y 473.784,Z 325.631,A -85,B 0,C 180,E1 -7287.448,E2 -7287.448} C_VEL
LIN {X 0,Y 473.758,Z 326.675,A -85,B 0,C 180,E1 -7288.299,E2 -7288.299} C_VEL
LIN {X 0,Y 473.696,Z 327.317,A -85,B 0,C 180,E1 -7289.149,E2 -7289.149} C_VEL
LIN {X 0,Y 473.683,Z 327.555,A -85,B 0,C 180,E1 -7289.999,E2 -7289.999} C_VEL
LIN {X 0,Y 473.695,Z 327.342,A -85,B 0,C 180,E1 -7290.849,E2 -7290.849} C_VEL
LIN {X 0,Y 473.758,Z 326.732,A -85,B 0,C 180,E1 -7291.699,E2 -7291.699} C_VEL
LIN {X 0,Y 473.783,Z 325.721,A -85,B 0,C 180,E1 -7292.549,E2 -7292.549} C_VEL
LIN {X 0,Y 473.82,Z 324.259,A -85,B 0,C 180,E1 -7293.4,E2 -7293.4} C_VEL
LIN {X 0,Y 473.764,Z 321.219,A -85,B 0,C 180,E1 -7294.679,E2 -7294.679} C_VEL
LIN {X 0,Y 473.834,Z 317.089,A -85,B 0,C 180,E1 -7295.958,E2 -7295.958} C_VEL
LIN {X 0,Y 473.999,Z 310.731,A -85,B 0,C 180,E1 -7297.453,E2 -7297.453} C_VEL
LIN {X 0,Y 474.157,Z 303.758,A -85,B 0,C 180,E1 -7298.737,E2 -7298.737} C_VEL
LIN {X 0,Y 474.431,Z 294.959,A -85,B 0,C 180,E1 -7300.022,E2 -7300.022} C_VEL
LIN {X 0,Y 474.865,Z 284.928,A -85,B 0,C 180,E1 -7301.199,E2 -7301.199} C_VEL
LIN {X 0,Y 475.209,Z 275.34,A -85,B 0,C 180,E1 -7302.104,E2 -7302.104} C_VEL
LIN {X 0,Y 475.603,Z 263.149,A -85,B 0,C 180,E1 -7303.022,E2 -7303.022} C_VEL
LIN {X 0,Y 475.998,Z 251.094,A -85,B 0,C 180,E1 -7303.717,E2 -7303.717} C_VEL
LIN {X 0,Y 476.35,Z 237.715,A -85,B 0,C 180,E1 -7304.279,E2 -7304.279} C_VEL
LIN {X 0,Y 475.942,Z 231.64,A -85,B 0,C 180,E1 -7304.482,E2 -7304.482} C_VEL
LIN {X 0,Y 474.599,Z 220.616,A -85,B 0,C 180,E1 -7304.771,E2 -7304.771} C_VEL
LIN {X 0,Y 475.136,Z 205.788,A -85,B 0,C 180,E1 -7308.095,E2 -7308.095} C_VEL
LIN {X 0,Y 475.8,Z 190.164,A -85,B 0,C 180,E1 -7311.669,E2 -7311.669} C_VEL
LIN {X 0,Y 476.547,Z 176.558,A -85,B 0,C 180,E1 -7314.852,E2 -7314.852} C_VEL
LIN {X 0,Y 477.09,Z 166.872,A -85,B 0,C 180,E1 -7317.17,E2 -7317.17} C_VEL
LIN {X 0,Y 476.172,Z 161.031,A -85,B 0,C 180,E1 -7318.663,E2 -7318.663} C_VEL
LIN {X 0,Y 474.602,Z 153.37,A -85,B 0,C 180,E1 -7320.729,E2 -7320.729} C_VEL
LIN {X 0,Y 474.637,Z 153.362,A -85,B 0,C 180,E1 -7323.218,E2 -7323.218} C_VEL
LIN {X 0,Y 474.587,Z 153.369,A -85,B 0,C 180,E1 -7326.321,E2 -7326.321} C_VEL
LIN {X 0,Y 474.617,Z 153.364,A -85,B 0,C 180,E1 -7329.546,E2 -7329.546} C_VEL
LIN {X 0,Y 474.591,Z 153.368,A -85,B 0,C 180,E1 -7332.232,E2 -7332.232} C_VEL
LIN {X 0,Y 474.612,Z 153.365,A -85,B 0,C 180,E1 -7335.296,E2 -7335.296} C_VEL
LIN {X 0,Y 474.629,Z 153.363,A -85,B 0,C 180,E1 -7338.215,E2 -7338.215} C_VEL
LIN {X 0,Y 474.663,Z 153.36,A -85,B 0,C 180,E1 -7340.456,E2 -7340.456} C_VEL
LIN {X 0,Y 474.572,Z 153.369,A -85,B 0,C 180,E1 -7343.675,E2 -7343.675} C_VEL
LIN {X 0,Y 474.631,Z 153.361,A -85,B 0,C 180,E1 -7346.779,E2 -7346.779} C_VEL
LIN {X 0,Y 474.602,Z 153.367,A -85,B 0,C 180,E1 -7349.769,E2 -7349.769} C_VEL
LIN {X 0,Y 474.702,Z 153.355,A -85,B 0,C 180,E1 -7352.68,E2 -7352.68} C_VEL
LIN {X 0,Y 474.638,Z 153.361,A -85,B 0,C 180,E1 -7355.506,E2 -7355.506} C_VEL
LIN {X 0,Y 474.656,Z 153.361,A -85,B 0,C 180,E1 -7359.185,E2 -7359.185} C_VEL
LIN {X 0,Y 474.643,Z 153.361,A -85,B 0,C 180,E1 -7361.884,E2 -7361.884} C_VEL
LIN {X 0,Y 474.685,Z 153.357,A -85,B 0,C 180,E1 -7364.544,E2 -7364.544} C_VEL
LIN {X 0,Y 474.723,Z 153.351,A -85,B 0,C 180,E1 -7368.038,E2 -7368.038} C_VEL
LIN {X 0,Y 474.71,Z 153.353,A -85,B 0,C 180,E1 -7371.486,E2 -7371.486} C_VEL
LIN {X 0,Y 474.769,Z 153.347,A -85,B 0,C 180,E1 -7374.052,E2 -7374.052} C_VEL
LIN {X 0,Y 474.882,Z 153.333,A -85,B 0,C 180,E1 -7377.455,E2 -7377.455} C_VEL
LIN {X 0,Y 474.894,Z 153.33,A -85,B 0,C 180,E1 -7380,E2 -7380} C_VEL
LIN {X 0,Y 474.873,Z 153.333,A -85,B 0,C 180,E1 -7382.545,E2 -7382.545} C_VEL
LIN {X 0,Y 474.764,Z 153.347,A -85,B 0,C 180,E1 -7385.948,E2 -7385.948} C_VEL
LIN {X 0,Y 474.715,Z 153.352,A -85,B 0,C 180,E1 -7388.514,E2 -7388.514} C_VEL
LIN {X 0,Y 474.724,Z 153.35,A -85,B 0,C 180,E1 -7391.962,E2 -7391.962} C_VEL
LIN {X 0,Y 474.666,Z 153.357,A -85,B 0,C 180,E1 -7395.768,E2 -7395.768} C_VEL
LIN {X 0,Y 474.651,Z 153.36,A -85,B 0,C 180,E1 -7399.011,E2 -7399.011} C_VEL
LIN {X 0,Y 474.623,Z 153.365,A -85,B 0,C 180,E1 -7401.727,E2 -7401.727} C_VEL
LIN {X 0,Y 474.641,Z 153.365,A -85,B 0,C 180,E1 -7404.494,E2 -7404.494} C_VEL
LIN {X 0,Y 474.622,Z 153.361,A -85,B 0,C 180,E1 -7407.325,E2 -7407.325} C_VEL
LIN {X 0,Y 474.591,Z 153.367,A -85,B 0,C 180,E1 -7410.231,E2 -7410.231} C_VEL
LIN {X 0,Y 474.631,Z 153.365,A -85,B 0,C 180,E1 -7413.221,E2 -7413.221} C_VEL
LIN {X 0,Y 474.582,Z 153.371,A -85,B 0,C 180,E1 -7416.324,E2 -7416.324} C_VEL
LIN {X 0,Y 474.616,Z 153.367,A -85,B 0,C 180,E1 -7419.649,E2 -7419.649} C_VEL
LIN {X 0,Y 474.621,Z 153.365,A -85,B 0,C 180,E1 -7422.934,E2 -7422.934} C_VEL
LIN {X 0,Y 474.605,Z 153.366,A -85,B 0,C 180,E1 -7425.897,E2 -7425.897} C_VEL
LIN {X 0,Y 474.624,Z 153.363,A -85,B 0,C 180,E1 -7429.041,E2 -7429.041} C_VEL
LIN {X 0,Y 474.6,Z 153.367,A -85,B 0,C 180,E1 -7431.706,E2 -7431.706} C_VEL
LIN {X 0,Y 474.615,Z 153.366,A -85,B 0,C 180,E1 -7434.727,E2 -7434.727} C_VEL
LIN {X 0,Y 474.632,Z 153.364,A -85,B 0,C 180,E1 -7437.79,E2 -7437.79} C_VEL
LIN {X 0,Y 474.626,Z 153.363,A -85,B 0,C 180,E1 -7440.884,E2 -7440.884} C_VEL
LIN {X 0,Y 474.623,Z 153.363,A -85,B 0,C 180,E1 -7443.628,E2 -7443.628} C_VEL
LIN {X 0,Y 474.63,Z 153.367,A -85,B 0,C 180,E1 -7446.644,E2 -7446.644} C_VEL
LIN {X 0,Y 474.652,Z 153.362,A -85,B 0,C 180,E1 -7450.091,E2 -7450.091} C_VEL
LIN {X 0,Y 474.653,Z 153.361,A -85,B 0,C 180,E1 -7451.694,E2 -7451.694} C_VEL
LIN {X 0,Y 473.991,Z 153.445,A -85,B 0,C 180,E1 -7452.403,E2 -7452.403} C_VEL
LIN {X 0,Y 471.138,Z 153.802,A -85,B 0,C 180,E1 -7453.554,E2 -7453.554} C_VEL
LIN {X 0,Y 468.719,Z 154.102,A -85,B 0,C 180,E1 -7454.483,E2 -7454.483} C_VEL
LIN {X 0,Y 467.676,Z 154.23,A -85,B 0,C 180,E1 -7455.2,E2 -7455.2} C_VEL
LIN {X 0,Y 467.59,Z 154.239,A -85,B 0,C 180,E1 -7455.443,E2 -7455.443} C_VEL
LIN {X 0,Y 467.649,Z 154.232,A -85,B 0,C 180,E1 -7458.735,E2 -7458.735} C_VEL
LIN {X 0,Y 467.749,Z 154.221,A -85,B 0,C 180,E1 -7462.23,E2 -7462.23} C_VEL
LIN {X 0,Y 467.725,Z 154.225,A -85,B 0,C 180,E1 -7464.829,E2 -7464.829} C_VEL
LIN {X 0,Y 467.861,Z 154.206,A -85,B 0,C 180,E1 -7467.418,E2 -7467.418} C_VEL
LIN {X 0,Y 467.851,Z 154.21,A -85,B 0,C 180,E1 -7470.001,E2 -7470.001} C_VEL
LIN {X 0,Y 467.852,Z 154.206,A -85,B 0,C 180,E1 -7472.584,E2 -7472.584} C_VEL
LIN {X 0,Y 467.746,Z 154.22,A -85,B 0,C 180,E1 -7476.039,E2 -7476.039} C_VEL
LIN {X 0,Y 467.683,Z 154.229,A -85,B 0,C 180,E1 -7478.644,E2 -7478.644} C_VEL
LIN {X 0,Y 467.658,Z 154.23,A -85,B 0,C 180,E1 -7482.359,E2 -7482.359} C_VEL
LIN {X 0,Y 467.653,Z 154.231,A -85,B 0,C 180,E1 -7485.886,E2 -7485.886} C_VEL
LIN {X 0,Y 467.627,Z 154.235,A -85,B 0,C 180,E1 -7489.309,E2 -7489.309} C_VEL
LIN {X 0,Y 467.538,Z 154.247,A -85,B 0,C 180,E1 -7492.075,E2 -7492.075} C_VEL
LIN {X 0,Y 467.563,Z 154.243,A -85,B 0,C 180,E1 -7494.891,E2 -7494.891} C_VEL
LIN {X 0,Y 467.55,Z 154.243,A -85,B 0,C 180,E1 -7497.775,E2 -7497.775} C_VEL
LIN {X 0,Y 467.57,Z 154.242,A -85,B 0,C 180,E1 -7501.045,E2 -7501.045} C_VEL
LIN {X 0,Y 467.582,Z 154.241,A -85,B 0,C 180,E1 -7504.241,E2 -7504.241} C_VEL
LIN {X 0,Y 467.526,Z 154.249,A -85,B 0,C 180,E1 -7507.183,E2 -7507.183} C_VEL
LIN {X 0,Y 467.562,Z 154.245,A -85,B 0,C 180,E1 -7510.267,E2 -7510.267} C_VEL
LIN {X 0,Y 467.548,Z 154.246,A -85,B 0,C 180,E1 -7512.566,E2 -7512.566} C_VEL
LIN {X 0,Y 467.571,Z 154.244,A -85,B 0,C 180,E1 -7515.053,E2 -7515.053} C_VEL
LIN {X 0,Y 467.594,Z 154.24,A -85,B 0,C 180,E1 -7517.44,E2 -7517.44} C_VEL
LIN {X 0,Y 467.553,Z 154.243,A -85,B 0,C 180,E1 -7520.852,E2 -7520.852} C_VEL
LIN {X 0,Y 467.56,Z 154.244,A -85,B 0,C 180,E1 -7524.262,E2 -7524.262} C_VEL
LIN {X 0,Y 467.598,Z 154.243,A -85,B 0,C 180,E1 -7527.319,E2 -7527.319} C_VEL
LIN {X 0,Y 467.649,Z 154.36,A -85,B 0,C 180,E1 -7528.011,E2 -7528.011} C_VEL
LIN {X 0,Y 468.328,Z 158.813,A -85,B 0,C 180,E1 -7529.82,E2 -7529.82} C_VEL
LIN {X 0,Y 468.09,Z 166.433,A -85,B 0,C 180,E1 -7532.786,E2 -7532.786} C_VEL
LIN {X 0,Y 467.784,Z 175.034,A -85,B 0,C 180,E1 -7536.068,E2 -7536.068} C_VEL
LIN {X 0,Y 467.552,Z 183.659,A -85,B 0,C 180,E1 -7539.314,E2 -7539.314} C_VEL
LIN {X 0,Y 467.304,Z 192.271,A -85,B 0,C 180,E1 -7542.495,E2 -7542.495} C_VEL
LIN {X 0,Y 467.143,Z 200.828,A -85,B 0,C 180,E1 -7545.627,E2 -7545.627} C_VEL
LIN {X 0,Y 466.968,Z 209.392,A -85,B 0,C 180,E1 -7548.717,E2 -7548.717} C_VEL
LIN {X 0,Y 466.878,Z 215.056,A -85,B 0,C 180,E1 -7550.742,E2 -7550.742} C_VEL
LIN {X 0,Y 468,Z 225.137,A -85,B 0,C 180,E1 -7551.2,E2 -7551.2} C_VEL
LIN {X 0,Y 467.973,Z 233.392,A -85,B 0,C 180,E1 -7551.689,E2 -7551.689} C_VEL
LIN {X 0,Y 467.686,Z 241.934,A -85,B 0,C 180,E1 -7552.347,E2 -7552.347} C_VEL
LIN {X 0,Y 467.483,Z 249.458,A -85,B 0,C 180,E1 -7553.092,E2 -7553.092} C_VEL
LIN {X 0,Y 467.267,Z 256.353,A -85,B 0,C 180,E1 -7553.956,E2 -7553.956} C_VEL
LIN {X 0,Y 467.175,Z 263.004,A -85,B 0,C 180,E1 -7555.038,E2 -7555.038} C_VEL
LIN {X 0,Y 467.014,Z 267.983,A -85,B 0,C 180,E1 -7556.117,E2 -7556.117} C_VEL
LIN {X 0,Y 466.811,Z 272.187,A -85,B 0,C 180,E1 -7557.411,E2 -7557.411} C_VEL
LIN {X 0,Y 466.713,Z 274.04,A -85,B 0,C 180,E1 -7558.274,E2 -7558.274} C_VEL
LIN {X 0,Y 466.645,Z 275.192,A -85,B 0,C 180,E1 -7559.137,E2 -7559.137} C_VEL
LIN {X 0,Y 466.629,Z 275.666,A -85,B 0,C 180,E1 -7560,E2 -7560} C_VEL
LIN {X 0,Y 466.646,Z 275.469,A -85,B 0,C 180,E1 -7560.863,E2 -7560.863} C_VEL
LIN {X 0,Y 466.716,Z 274.6,A -85,B 0,C 180,E1 -7561.726,E2 -7561.726} C_VEL
LIN {X 0,Y 466.923,Z 271.998,A -85,B 0,C 180,E1 -7563.02,E2 -7563.02} C_VEL
LIN {X 0,Y 467.097,Z 269.332,A -85,B 0,C 180,E1 -7563.882,E2 -7563.882} C_VEL
LIN {X 0,Y 467.225,Z 264.824,A -85,B 0,C 180,E1 -7564.962,E2 -7564.962} C_VEL
LIN {X 0,Y 467.298,Z 258.798,A -85,B 0,C 180,E1 -7566.043,E2 -7566.043} C_VEL
LIN {X 0,Y 467.598,Z 251.464,A -85,B 0,C 180,E1 -7567.042,E2 -7567.042} C_VEL
LIN {X 0,Y 467.959,Z 243.514,A -85,B 0,C 180,E1 -7567.877,E2 -7567.877} C_VEL
LIN {X 0,Y 468.384,Z 234.161,A -85,B 0,C 180,E1 -7568.63,E2 -7568.63} C_VEL
LIN {X 0,Y 468.362,Z 225.411,A -85,B 0,C 180,E1 -7569.174,E2 -7569.174} C_VEL
LIN {X 0,Y 467.017,Z 215.612,A -85,B 0,C 180,E1 -7569.692,E2 -7569.692} C_VEL
LIN {X 0,Y 467.167,Z 207.705,A -85,B 0,C 180,E1 -7572.6,E2 -7572.6} C_VEL
LIN {X 0,Y 467.419,Z 199.156,A -85,B 0,C 180,E1 -7575.783,E2 -7575.783} C_VEL
LIN {X 0,Y 467.667,Z 191.291,A -85,B 0,C 180,E1 -7578.78,E2 -7578.78} C_VEL
LIN {X 0,Y 467.948,Z 182.889,A -85,B 0,C 180,E1 -7582.053,E2 -7582.053} C_VEL
LIN {X 0,Y 468.266,Z 175.93,A -85,B 0,C 180,E1 -7584.85,E2 -7584.85} C_VEL
LIN {X 0,Y 468.777,Z 168.865,A -85,B 0,C 180,E1 -7587.804,E2 -7587.804} C_VEL
LIN {X 0,Y 469.089,Z 163.512,A -85,B 0,C 180,E1 -7590.126,E2 -7590.126} C_VEL
LIN {X 0,Y 468.617,Z 159.304,A -85,B 0,C 180,E1 -7592.168,E2 -7592.168} C_VEL
LIN {X 0,Y 467.593,Z 154.243,A -85,B 0,C 180,E1 -7594.962,E2 -7594.962} C_VEL
LIN {X 0,Y 467.568,Z 154.246,A -85,B 0,C 180,E1 -7598.59,E2 -7598.59} C_VEL
LIN {X 0,Y 467.582,Z 154.245,A -85,B 0,C 180,E1 -7601.403,E2 -7601.403} C_VEL
LIN {X 0,Y 467.555,Z 154.247,A -85,B 0,C 180,E1 -7603.82,E2 -7603.82} C_VEL
LIN {X 0,Y 467.56,Z 154.246,A -85,B 0,C 180,E1 -7606.255,E2 -7606.255} C_VEL
LIN {X 0,Y 467.584,Z 154.243,A -85,B 0,C 180,E1 -7608.723,E2 -7608.723} C_VEL
LIN {X 0,Y 467.571,Z 154.245,A -85,B 0,C 180,E1 -7611.955,E2 -7611.955} C_VEL
LIN {X 0,Y 467.564,Z 154.246,A -85,B 0,C 180,E1 -7615.166,E2 -7615.166} C_VEL
LIN {X 0,Y 467.6,Z 154.299,A -85,B 0,C 180,E1 -7616.099,E2 -7616.099} C_VEL
LIN {X 0,Y 468.944,Z 160.222,A -85,B 0,C 180,E1 -7618.678,E2 -7618.678} C_VEL
LIN {X 0,Y 470.51,Z 167.783,A -85,B 0,C 180,E1 -7621.445,E2 -7621.445} C_VEL
LIN {X 0,Y 470.905,Z 170.877,A -85,B 0,C 180,E1 -7622.44,E2 -7622.44} C_VEL
LIN {X 0,Y 470.296,Z 177.403,A -85,B 0,C 180,E1 -7624.317,E2 -7624.317} C_VEL
LIN {X 0,Y 469.318,Z 187.733,A -85,B 0,C 180,E1 -7627.085,E2 -7627.085} C_VEL
LIN {X 0,Y 468.47,Z 200.453,A -85,B 0,C 180,E1 -7630.271,E2 -7630.271} C_VEL
LIN {X 0,Y 467.829,Z 213.653,A -85,B 0,C 180,E1 -7633.414,E2 -7633.414} C_VEL
LIN {X 0,Y 467.578,Z 220.597,A -85,B 0,C 180,E1 -7635.013,E2 -7635.013} C_VEL
LIN {X 0,Y 469.124,Z 233.296,A -85,B 0,C 180,E1 -7635.383,E2 -7635.383} C_VEL
LIN {X 0,Y 469.334,Z 240.366,A -85,B 0,C 180,E1 -7635.639,E2 -7635.639} C_VEL
LIN {X 0,Y 468.961,Z 253.217,A -85,B 0,C 180,E1 -7636.236,E2 -7636.236} C_VEL
LIN {X 0,Y 468.502,Z 265.411,A -85,B 0,C 180,E1 -7636.995,E2 -7636.995} C_VEL
LIN {X 0,Y 468.108,Z 276.275,A -85,B 0,C 180,E1 -7637.865,E2 -7637.865} C_VEL
LIN {X 0,Y 467.7,Z 287.086,A -85,B 0,C 180,E1 -7638.953,E2 -7638.953} C_VEL
LIN {X 0,Y 467.328,Z 295.845,A -85,B 0,C 180,E1 -7640.04,E2 -7640.04} C_VEL
LIN {X 0,Y 467.076,Z 304.316,A -85,B 0,C 180,E1 -7641.345,E2 -7641.345} C_VEL
LIN {X 0,Y 466.855,Z 311.107,A -85,B 0,C 180,E1 -7642.647,E2 -7642.647} C_VEL
LIN {X 0,Y 466.741,Z 316.504,A -85,B 0,C 180,E1 -7643.948,E2 -7643.948} C_VEL
LIN {X 0,Y 466.697,Z 320.681,A -85,B 0,C 180,E1 -7645.248,E2 -7645.248} C_VEL
LIN {X 0,Y 466.731,Z 323.761,A -85,B 0,C 180,E1 -7646.546,E2 -7646.546} C_VEL
LIN {X 0,Y 466.702,Z 325.242,A -85,B 0,C 180,E1 -7647.409,E2 -7647.409} C_VEL
LIN {X 0,Y 466.693,Z 326.288,A -85,B 0,C 180,E1 -7648.273,E2 -7648.273} C_VEL
LIN {X 0,Y 466.627,Z 326.93,A -85,B 0,C 180,E1 -7649.136,E2 -7649.136} C_VEL
LIN {X 0,Y 466.612,Z 327.163,A -85,B 0,C 180,E1 -7649.999,E2 -7649.999} C_VEL
LIN {X 0,Y 466.693,Z 326.331,A -85,B 0,C 180,E1 -7651.725,E2 -7651.725} C_VEL
LIN {X 0,Y 466.701,Z 325.312,A -85,B 0,C 180,E1 -7652.588,E2 -7652.588} C_VEL
LIN {X 0,Y 466.728,Z 323.833,A -85,B 0,C 180,E1 -7653.452,E2 -7653.452} C_VEL
LIN {X 0,Y 466.692,Z 320.774,A -85,B 0,C 180,E1 -7654.75,E2 -7654.75} C_VEL
LIN {X 0,Y 466.75,Z 316.617,A -85,B 0,C 180,E1 -7656.049,E2 -7656.049} C_VEL
LIN {X 0,Y 466.904,Z 310.228,A -85,B 0,C 180,E1 -7657.567,E2 -7657.567} C_VEL
LIN {X 0,Y 467.091,Z 303.202,A -85,B 0,C 180,E1 -7658.87,E2 -7658.87} C_VEL
LIN {X 0,Y 467.402,Z 294.347,A -85,B 0,C 180,E1 -7660.175,E2 -7660.175} C_VEL
LIN {X 0,Y 467.784,Z 285.241,A -85,B 0,C 180,E1 -7661.261,E2 -7661.261} C_VEL
LIN {X 0,Y 468.209,Z 274.826,A -85,B 0,C 180,E1 -7662.263,E2 -7662.263} C_VEL
LIN {X 0,Y 468.56,Z 263.795,A -85,B 0,C 180,E1 -7663.111,E2 -7663.111} C_VEL
LIN {X 0,Y 468.983,Z 252.064,A -85,B 0,C 180,E1 -7663.816,E2 -7663.816} C_VEL
LIN {X 0,Y 469.324,Z 239.877,A -85,B 0,C 180,E1 -7664.359,E2 -7664.359} C_VEL
LIN {X 0,Y 469.189,Z 234.311,A -85,B 0,C 180,E1 -7664.557,E2 -7664.557} C_VEL
LIN {X 0,Y 467.542,Z 220.57,A -85,B 0,C 180,E1 -7664.943,E2 -7664.943} C_VEL
LIN {X 0,Y 468.134,Z 205.544,A -85,B 0,C 180,E1 -7668.375,E2 -7668.375} C_VEL
LIN {X 0,Y 468.761,Z 191.547,A -85,B 0,C 180,E1 -7671.635,E2 -7671.635} C_VEL
LIN {X 0,Y 469.549,Z 178.352,A -85,B 0,C 180,E1 -7674.775,E2 -7674.775} C_VEL
LIN {X 0,Y 470.12,Z 168.661,A -85,B 0,C 180,E1 -7677.125,E2 -7677.125} C_VEL
LIN {X 0,Y 469.597,Z 164.21,A -85,B 0,C 180,E1 -7678.272,E2 -7678.272} C_VEL
LIN {X 0,Y 467.558,Z 154.247,A -85,B 0,C 180,E1 -7680.962,E2 -7680.962} C_VEL
LIN {X 0,Y 467.585,Z 154.244,A -85,B 0,C 180,E1 -7684.241,E2 -7684.241} C_VEL
LIN {X 0,Y 467.543,Z 154.248,A -85,B 0,C 180,E1 -7687.185,E2 -7687.185} C_VEL
LIN {X 0,Y 467.561,Z 154.243,A -85,B 0,C 180,E1 -7690.264,E2 -7690.264} C_VEL
LIN {X 0,Y 467.541,Z 154.245,A -85,B 0,C 180,E1 -7693.744,E2 -7693.744} C_VEL
LIN {X 0,Y 467.568,Z 154.244,A -85,B 0,C 180,E1 -7696.257,E2 -7696.257} C_VEL
LIN {X 0,Y 467.579,Z 154.242,A -85,B 0,C 180,E1 -7698.72,E2 -7698.72} C_VEL
LIN {X 0,Y 467.566,Z 154.243,A -85,B 0,C 180,E1 -7701.406,E2 -7701.406} C_VEL
LIN {X 0,Y 467.545,Z 154.249,A -85,B 0,C 180,E1 -7704.26,E2 -7704.26} C_VEL
LIN {X 0,Y 467.57,Z 154.242,A -85,B 0,C 180,E1 -7707.32,E2 -7707.32} C_VEL
LIN {X 0,Y 467.566,Z 154.245,A -85,B 0,C 180,E1 -7710.664,E2 -7710.664} C_VEL
LIN {X 0,Y 467.613,Z 154.237,A -85,B 0,C 180,E1 -7713.199,E2 -7713.199} C_VEL
LIN {X 0,Y 467.578,Z 154.24,A -85,B 0,C 180,E1 -7716.468,E2 -7716.468} C_VEL
LIN {X 0,Y 467.609,Z 154.238,A -85,B 0,C 180,E1 -7719.776,E2 -7719.776} C_VEL
LIN {X 0,Y 467.596,Z 154.24,A -85,B 0,C 180,E1 -7722.506,E2 -7722.506} C_VEL
LIN {X 0,Y 467.592,Z 154.239,A -85,B 0,C 180,E1 -7725.196,E2 -7725.196} C_VEL
LIN {X 0,Y 467.666,Z 154.231,A -85,B 0,C 180,E1 -7727.855,E2 -7727.855} C_VEL
LIN {X 0,Y 467.663,Z 154.232,A -85,B 0,C 180,E1 -7731.357,E2 -7731.357} C_VEL
LIN {X 0,Y 467.733,Z 154.223,A -85,B 0,C 180,E1 -7733.962,E2 -7733.962} C_VEL
LIN {X 0,Y 467.847,Z 154.209,A -85,B 0,C 180,E1 -7737.417,E2 -7737.417} C_VEL
LIN {X 0,Y 467.865,Z 154.205,A -85,B 0,C 180,E1 -7740,E2 -7740} C_VEL
LIN {X 0,Y 467.839,Z 154.209,A -85,B 0,C 180,E1 -7742.583,E2 -7742.583} C_VEL
LIN {X 0,Y 467.728,Z 154.223,A -85,B 0,C 180,E1 -7746.038,E2 -7746.038} C_VEL
LIN {X 0,Y 467.668,Z 154.23,A -85,B 0,C 180,E1 -7748.643,E2 -7748.643} C_VEL
LIN {X 0,Y 467.668,Z 154.229,A -85,B 0,C 180,E1 -7752.145,E2 -7752.145} C_VEL
LIN {X 0,Y 467.634,Z 154.233,A -85,B 0,C 180,E1 -7755.886,E2 -7755.886} C_VEL
LIN {X 0,Y 467.61,Z 154.238,A -85,B 0,C 180,E1 -7759.308,E2 -7759.308} C_VEL
LIN {X 0,Y 467.553,Z 154.244,A -85,B 0,C 180,E1 -7762.073,E2 -7762.073} C_VEL
LIN {X 0,Y 467.58,Z 154.241,A -85,B 0,C 180,E1 -7764.889,E2 -7764.889} C_VEL
LIN {X 0,Y 467.566,Z 154.243,A -85,B 0,C 180,E1 -7767.773,E2 -7767.773} C_VEL
LIN {X 0,Y 467.557,Z 154.244,A -85,B 0,C 180,E1 -7771.046,E2 -7771.046} C_VEL
